LIN {X 0,Y 280.573,Z 825.158,A -85,B 0,C 180,E1 -18219.062,E2 -18219.062} C_VEL
LIN {X 0,Y 279.495,Z 836.896,A -85,B 0,C 180,E1 -18220.065,E2 -18220.065} C_VEL
LIN {X 0,Y 278.097,Z 847.663,A -85,B 0,C 180,E1 -18221.254,E2 -18221.254} C_VEL
LIN {X 0,Y 276.309,Z 858.858,A -85,B 0,C 180,E1 -18222.844,E2 -18222.844} C_VEL
LIN {X 0,Y 274.292,Z 869.192,A -85,B 0,C 180,E1 -18224.686,E2 -18224.686} C_VEL
LIN {X 0,Y 272.634,Z 876.745,A -85,B 0,C 180,E1 -18226.359,E2 -18226.359} C_VEL
LIN {X 0,Y 270.784,Z 884.275,A -85,B 0,C 180,E1 -18228.399,E2 -18228.399} C_VEL
LIN {X 0,Y 269.028,Z 890.984,A -85,B 0,C 180,E1 -18230.695,E2 -18230.695} C_VEL
LIN {X 0,Y 267.576,Z 895.963,A -85,B 0,C 180,E1 -18232.839,E2 -18232.839} C_VEL
LIN {X 0,Y 266.081,Z 900.757,A -85,B 0,C 180,E1 -18235.569,E2 -18235.569} C_VEL
LIN {X 0,Y 265.124,Z 903.749,A -85,B 0,C 180,E1 -18238.025,E2 -18238.025} C_VEL
LIN {X 0,Y 264.627,Z 905.127,A -85,B 0,C 180,E1 -18239.698,E2 -18239.698} C_VEL
LIN {X 0,Y 264.256,Z 906.046,A -85,B 0,C 180,E1 -18241.401,E2 -18241.401} C_VEL
LIN {X 0,Y 263.97,Z 906.49,A -85,B 0,C 180,E1 -18243.091,E2 -18243.091} C_VEL
LIN {X 0,Y 263.816,Z 906.395,A -85,B 0,C 180,E1 -18244.926,E2 -18244.926} C_VEL
LIN {X 0,Y 263.785,Z 905.92,A -85,B 0,C 180,E1 -18246.447,E2 -18246.447} C_VEL
LIN {X 0,Y 263.951,Z 904.438,A -85,B 0,C 180,E1 -18248.737,E2 -18248.737} C_VEL
LIN {X 0,Y 264.462,Z 901.575,A -85,B 0,C 180,E1 -18251.406,E2 -18251.406} C_VEL
LIN {X 0,Y 265.271,Z 897.734,A -85,B 0,C 180,E1 -18253.851,E2 -18253.851} C_VEL
LIN {X 0,Y 266.194,Z 892.722,A -85,B 0,C 180,E1 -18256.257,E2 -18256.257} C_VEL
LIN {X 0,Y 267.446,Z 886.349,A -85,B 0,C 180,E1 -18258.636,E2 -18258.636} C_VEL
LIN {X 0,Y 268.929,Z 878.429,A -85,B 0,C 180,E1 -18260.981,E2 -18260.981} C_VEL
LIN {X 0,Y 270.327,Z 870.307,A -85,B 0,C 180,E1 -18262.909,E2 -18262.909} C_VEL
LIN {X 0,Y 271.929,Z 860.358,A -85,B 0,C 180,E1 -18264.812,E2 -18264.812} C_VEL
LIN {X 0,Y 273.479,Z 849.327,A -85,B 0,C 180,E1 -18266.503,E2 -18266.503} C_VEL
LIN {X 0,Y 274.856,Z 837.273,A -85,B 0,C 180,E1 -18267.939,E2 -18267.939} C_VEL
LIN {X 0,Y 275.911,Z 824.671,A -85,B 0,C 180,E1 -18269.09,E2 -18269.09} C_VEL
LIN {X 0,Y 276.523,Z 812.385,A -85,B 0,C 180,E1 -18269.911,E2 -18269.911} C_VEL
LIN {X 0,Y 276.817,Z 798.91,A -85,B 0,C 180,E1 -18270.5,E2 -18270.5} C_VEL
LIN {X 0,Y 277.725,Z 751.411,A -85,B 0,C 180,E1 -18271.806,E2 -18271.806} C_VEL
LIN {X 0,Y 271.657,Z 736.963,A -85,B 0,C 180,E1 -18272.837,E2 -18272.837} C_VEL
LIN {X 0,Y 264.688,Z 722.978,A -85,B 0,C 180,E1 -18273.994,E2 -18273.994} C_VEL
LIN {X 0,Y 263.476,Z 720.392,A -85,B 0,C 180,E1 -18274.273,E2 -18274.273} C_VEL
LIN {X 0,Y 263.344,Z 719.73,A -85,B 0,C 180,E1 -18274.594,E2 -18274.594} C_VEL
LIN {X 0,Y 263.53,Z 719.652,A -85,B 0,C 180,E1 -18277.665,E2 -18277.665} C_VEL
LIN {X 0,Y 263.339,Z 719.672,A -85,B 0,C 180,E1 -18280.769,E2 -18280.769} C_VEL
LIN {X 0,Y 263.315,Z 719.673,A -85,B 0,C 180,E1 -18285.482,E2 -18285.482} C_VEL
LIN {X 0,Y 263.214,Z 719.678,A -85,B 0,C 180,E1 -18290.313,E2 -18290.313} C_VEL
LIN {X 0,Y 263.127,Z 719.691,A -85,B 0,C 180,E1 -18295.302,E2 -18295.302} C_VEL
LIN {X 0,Y 263.124,Z 719.7,A -85,B 0,C 180,E1 -18298.739,E2 -18298.739} C_VEL
LIN {X 0,Y 263.133,Z 719.698,A -85,B 0,C 180,E1 -18302.291,E2 -18302.291} C_VEL
LIN {X 0,Y 263.163,Z 719.673,A -85,B 0,C 180,E1 -18305.984,E2 -18305.984} C_VEL
LIN {X 0,Y 263.097,Z 719.713,A -85,B 0,C 180,E1 -18309.877,E2 -18309.877} C_VEL
LIN {X 0,Y 263.083,Z 719.716,A -85,B 0,C 180,E1 -18313.995,E2 -18313.995} C_VEL
LIN {X 0,Y 263.087,Z 719.713,A -85,B 0,C 180,E1 -18318.419,E2 -18318.419} C_VEL
LIN {X 0,Y 263.211,Z 719.896,A -85,B 0,C 180,E1 -18321.285,E2 -18321.285} C_VEL
LIN {X 0,Y 263.406,Z 720.866,A -85,B 0,C 180,E1 -18321.514,E2 -18321.514} C_VEL
LIN {X 0,Y 272.271,Z 746.098,A -85,B 0,C 180,E1 -18323.036,E2 -18323.036} C_VEL
LIN {X 0,Y 270.678,Z 798.339,A -85,B 0,C 180,E1 -18324.909,E2 -18324.909} C_VEL
LIN {X 0,Y 270.307,Z 809.826,A -85,B 0,C 180,E1 -18325.528,E2 -18325.528} C_VEL
LIN {X 0,Y 269.831,Z 820.372,A -85,B 0,C 180,E1 -18326.292,E2 -18326.292} C_VEL
LIN {X 0,Y 269.164,Z 830.302,A -85,B 0,C 180,E1 -18327.194,E2 -18327.194} C_VEL
LIN {X 0,Y 268.375,Z 841.093,A -85,B 0,C 180,E1 -18328.416,E2 -18328.416} C_VEL
LIN {X 0,Y 267.591,Z 849.983,A -85,B 0,C 180,E1 -18329.63,E2 -18329.63} C_VEL
LIN {X 0,Y 266.8,Z 858.729,A -85,B 0,C 180,E1 -18331.051,E2 -18331.051} C_VEL
LIN {X 0,Y 266.128,Z 866.2,A -85,B 0,C 180,E1 -18332.474,E2 -18332.474} C_VEL
LIN {X 0,Y 265.279,Z 874.154,A -85,B 0,C 180,E1 -18334.262,E2 -18334.262} C_VEL
LIN {X 0,Y 264.643,Z 881.015,A -85,B 0,C 180,E1 -18336.109,E2 -18336.109} C_VEL
LIN {X 0,Y 264.127,Z 887.251,A -85,B 0,C 180,E1 -18338.129,E2 -18338.129} C_VEL
LIN {X 0,Y 263.808,Z 891.489,A -85,B 0,C 180,E1 -18339.737,E2 -18339.737} C_VEL
LIN {X 0,Y 263.602,Z 894.43,A -85,B 0,C 180,E1 -18341.058,E2 -18341.058} C_VEL
LIN {X 0,Y 262.845,Z 896.919,A -85,B 0,C 180,E1 -18342.214,E2 -18342.214} C_VEL
LIN {X 0,Y 259.935,Z 900.48,A -85,B 0,C 180,E1 -18344.142,E2 -18344.142} C_VEL
LIN {X 0,Y 257.584,Z 902.751,A -85,B 0,C 180,E1 -18345.754,E2 -18345.754} C_VEL
LIN {X 0,Y 256.67,Z 904.09,A -85,B 0,C 180,E1 -18347.027,E2 -18347.027} C_VEL
LIN {X 0,Y 256.645,Z 904.457,A -85,B 0,C 180,E1 -18347.461,E2 -18347.461} C_VEL
LIN {X 0,Y 257.147,Z 906.07,A -85,B 0,C 180,E1 -18349.717,E2 -18349.717} C_VEL
LIN {X 0,Y 257.916,Z 906.726,A -85,B 0,C 180,E1 -18352.169,E2 -18352.169} C_VEL
LIN {X 0,Y 258.537,Z 906.558,A -85,B 0,C 180,E1 -18353.757,E2 -18353.757} C_VEL
LIN {X 0,Y 259.369,Z 905.964,A -85,B 0,C 180,E1 -18355.337,E2 -18355.337} C_VEL
LIN {X 0,Y 261.321,Z 903.482,A -85,B 0,C 180,E1 -18358.459,E2 -18358.459} C_VEL
LIN {X 0,Y 263.036,Z 900.45,A -85,B 0,C 180,E1 -18360.765,E2 -18360.765} C_VEL
LIN {X 0,Y 265.108,Z 896.26,A -85,B 0,C 180,E1 -18363.039,E2 -18363.039} C_VEL
LIN {X 0,Y 267.118,Z 891.825,A -85,B 0,C 180,E1 -18364.905,E2 -18364.905} C_VEL
LIN {X 0,Y 269.683,Z 885.252,A -85,B 0,C 180,E1 -18367.111,E2 -18367.111} C_VEL
LIN {X 0,Y 271.595,Z 880.039,A -85,B 0,C 180,E1 -18368.557,E2 -18368.557} C_VEL
LIN {X 0,Y 274.067,Z 872.242,A -85,B 0,C 180,E1 -18370.341,E2 -18370.341} C_VEL
LIN {X 0,Y 276.149,Z 864.832,A -85,B 0,C 180,E1 -18371.747,E2 -18371.747} C_VEL
LIN {X 0,Y 278.356,Z 856.069,A -85,B 0,C 180,E1 -18373.134,E2 -18373.134} C_VEL
LIN {X 0,Y 280.318,Z 846.92,A -85,B 0,C 180,E1 -18374.334,E2 -18374.334} C_VEL
LIN {X 0,Y 281.972,Z 837.469,A -85,B 0,C 180,E1 -18375.356,E2 -18375.356} C_VEL
LIN {X 0,Y 283.26,Z 827.918,A -85,B 0,C 180,E1 -18376.208,E2 -18376.208} C_VEL
LIN {X 0,Y 284.446,Z 816.78,A -85,B 0,C 180,E1 -18376.969,E2 -18376.969} C_VEL
LIN {X 0,Y 285.631,Z 800.883,A -85,B 0,C 180,E1 -18377.784,E2 -18377.784} C_VEL
LIN {X 0,Y 288.129,Z 773.827,A -85,B 0,C 180,E1 -18378.908,E2 -18378.908} C_VEL
LIN {X 0,Y 288.719,Z 767.247,A -85,B 0,C 180,E1 -18379.186,E2 -18379.186} C_VEL
LIN {X 0,Y 284.14,Z 758.529,A -85,B 0,C 180,E1 -18381.12,E2 -18381.12} C_VEL
LIN {X 0,Y 279.969,Z 751.63,A -85,B 0,C 180,E1 -18383.109,E2 -18383.109} C_VEL
LIN {X 0,Y 276.835,Z 747.044,A -85,B 0,C 180,E1 -18384.822,E2 -18384.822} C_VEL
LIN {X 0,Y 274.47,Z 743.25,A -85,B 0,C 180,E1 -18386.379,E2 -18386.379} C_VEL
LIN {X 0,Y 271.752,Z 740.074,A -85,B 0,C 180,E1 -18388.36,E2 -18388.36} C_VEL
LIN {X 0,Y 270.817,Z 738.098,A -85,B 0,C 180,E1 -18389.329,E2 -18389.329} C_VEL
LIN {X 0,Y 268.084,Z 735.681,A -85,B 0,C 180,E1 -18392.341,E2 -18392.341} C_VEL
LIN {X 0,Y 267.252,Z 733.95,A -85,B 0,C 180,E1 -18394.207,E2 -18394.207} C_VEL
LIN {X 0,Y 266.552,Z 733.96,A -85,B 0,C 180,E1 -18396.794,E2 -18396.794} C_VEL
LIN {X 0,Y 266.864,Z 735.363,A -85,B 0,C 180,E1 -18399.936,E2 -18399.936} C_VEL
LIN {X 0,Y 268.128,Z 737.207,A -85,B 0,C 180,E1 -18402.44,E2 -18402.44} C_VEL
LIN {X 0,Y 269.32,Z 739.283,A -85,B 0,C 180,E1 -18404.053,E2 -18404.053} C_VEL
LIN {X 0,Y 271.804,Z 742.654,A -85,B 0,C 180,E1 -18406.385,E2 -18406.385} C_VEL
LIN {X 0,Y 273.944,Z 746.353,A -85,B 0,C 180,E1 -18408.073,E2 -18408.073} C_VEL
LIN {X 0,Y 276.75,Z 755.997,A -85,B 0,C 180,E1 -18410.376,E2 -18410.376} C_VEL
LIN {X 0,Y 280.751,Z 769.642,A -85,B 0,C 180,E1 -18413.044,E2 -18413.044} C_VEL
LIN {X 0,Y 281.302,Z 772.583,A -85,B 0,C 180,E1 -18413.455,E2 -18413.455} C_VEL
LIN {X 0,Y 282.401,Z 792.767,A -85,B 0,C 180,E1 -18415.273,E2 -18415.273} C_VEL
LIN {X 0,Y 283.037,Z 812.394,A -85,B 0,C 180,E1 -18416.751,E2 -18416.751} C_VEL
LIN {X 0,Y 283.094,Z 822.192,A -85,B 0,C 180,E1 -18417.396,E2 -18417.396} C_VEL
LIN {X 0,Y 282.769,Z 841.316,A -85,B 0,C 180,E1 -18418.475,E2 -18418.475} C_VEL
LIN {X 0,Y 280.175,Z 867.058,A -85,B 0,C 180,E1 -18419.519,E2 -18419.519} C_VEL
LIN {X 0,Y 277.909,Z 882.038,A -85,B 0,C 180,E1 -18420.347,E2 -18420.347} C_VEL
LIN {X 0,Y 275.081,Z 895.368,A -85,B 0,C 180,E1 -18421.375,E2 -18421.375} C_VEL
LIN {X 0,Y 272.757,Z 905.306,A -85,B 0,C 180,E1 -18422.365,E2 -18422.365} C_VEL
LIN {X 0,Y 270.139,Z 915.057,A -85,B 0,C 180,E1 -18423.541,E2 -18423.541} C_VEL
LIN {X 0,Y 267.355,Z 924.567,A -85,B 0,C 180,E1 -18424.918,E2 -18424.918} C_VEL
LIN {X 0,Y 264.709,Z 933.598,A -85,B 0,C 180,E1 -18426.529,E2 -18426.529} C_VEL
LIN {X 0,Y 262.562,Z 940.532,A -85,B 0,C 180,E1 -18427.99,E2 -18427.99} C_VEL
LIN {X 0,Y 260.312,Z 948.007,A -85,B 0,C 180,E1 -18429.863,E2 -18429.863} C_VEL
LIN {X 0,Y 258.187,Z 955.518,A -85,B 0,C 180,E1 -18432.165,E2 -18432.165} C_VEL
LIN {X 0,Y 256.893,Z 960.781,A -85,B 0,C 180,E1 -18434.12,E2 -18434.12} C_VEL
LIN {X 0,Y 255.742,Z 965.991,A -85,B 0,C 180,E1 -18436.489,E2 -18436.489} C_VEL
LIN {X 0,Y 255.099,Z 970.126,A -85,B 0,C 180,E1 -18438.878,E2 -18438.878} C_VEL
LIN {X 0,Y 255.175,Z 976.468,A -85,B 0,C 180,E1 -18443.673,E2 -18443.673} C_VEL
LIN {X 0,Y 255.414,Z 978.203,A -85,B 0,C 180,E1 -18445.263,E2 -18445.263} C_VEL
LIN {X 0,Y 255.612,Z 979.494,A -85,B 0,C 180,E1 -18446.845,E2 -18446.845} C_VEL
LIN {X 0,Y 255.788,Z 980.353,A -85,B 0,C 180,E1 -18448.423,E2 -18448.423} C_VEL
LIN {X 0,Y 255.954,Z 980.742,A -85,B 0,C 180,E1 -18449.998,E2 -18449.998} C_VEL
LIN {X 0,Y 255.751,Z 980.652,A -85,B 0,C 180,E1 -18451.572,E2 -18451.572} C_VEL
LIN {X 0,Y 255.548,Z 980.148,A -85,B 0,C 180,E1 -18453.151,E2 -18453.151} C_VEL
LIN {X 0,Y 255.341,Z 979.232,A -85,B 0,C 180,E1 -18454.734,E2 -18454.734} C_VEL
LIN {X 0,Y 255.02,Z 976.923,A -85,B 0,C 180,E1 -18457.202,E2 -18457.202} C_VEL
LIN {X 0,Y 254.928,Z 973.806,A -85,B 0,C 180,E1 -18459.519,E2 -18459.519} C_VEL
LIN {X 0,Y 255.223,Z 969.585,A -85,B 0,C 180,E1 -18461.916,E2 -18461.916} C_VEL
LIN {X 0,Y 256.135,Z 963.256,A -85,B 0,C 180,E1 -18464.7,E2 -18464.7} C_VEL
LIN {X 0,Y 257.137,Z 957.383,A -85,B 0,C 180,E1 -18466.764,E2 -18466.764} C_VEL
LIN {X 0,Y 258.744,Z 951.013,A -85,B 0,C 180,E1 -18468.609,E2 -18468.609} C_VEL
LIN {X 0,Y 260.526,Z 943.101,A -85,B 0,C 180,E1 -18470.527,E2 -18470.527} C_VEL
LIN {X 0,Y 262.82,Z 933.587,A -85,B 0,C 180,E1 -18472.396,E2 -18472.396} C_VEL
LIN {X 0,Y 265.164,Z 923.078,A -85,B 0,C 180,E1 -18474.045,E2 -18474.045} C_VEL
LIN {X 0,Y 267.563,Z 911.507,A -85,B 0,C 180,E1 -18475.472,E2 -18475.472} C_VEL
LIN {X 0,Y 269.7,Z 899.511,A -85,B 0,C 180,E1 -18476.605,E2 -18476.605} C_VEL
LIN {X 0,Y 271.461,Z 886.354,A -85,B 0,C 180,E1 -18477.511,E2 -18477.511} C_VEL
LIN {X 0,Y 272.7,Z 872.76,A -85,B 0,C 180,E1 -18478.143,E2 -18478.143} C_VEL
LIN {X 0,Y 274.01,Z 835.757,A -85,B 0,C 180,E1 -18479.186,E2 -18479.186} C_VEL
LIN {X 0,Y 271.916,Z 808.359,A -85,B 0,C 180,E1 -18480.344,E2 -18480.344} C_VEL
LIN {X 0,Y 269.303,Z 784.538,A -85,B 0,C 180,E1 -18481.495,E2 -18481.495} C_VEL
LIN {X 0,Y 265.649,Z 760.465,A -85,B 0,C 180,E1 -18482.919,E2 -18482.919} C_VEL
LIN {X 0,Y 265.303,Z 757.226,A -85,B 0,C 180,E1 -18483.797,E2 -18483.797} C_VEL
LIN {X 0,Y 263.15,Z 746.364,A -85,B 0,C 180,E1 -18487.225,E2 -18487.225} C_VEL
LIN {X 0,Y 261.041,Z 737.55,A -85,B 0,C 180,E1 -18490.249,E2 -18490.249} C_VEL
LIN {X 0,Y 258.307,Z 728.035,A -85,B 0,C 180,E1 -18493.862,E2 -18493.862} C_VEL
LIN {X 0,Y 256.06,Z 720.679,A -85,B 0,C 180,E1 -18496.992,E2 -18496.992} C_VEL
LIN {X 0,Y 256.082,Z 720.572,A -85,B 0,C 180,E1 -18500.86,E2 -18500.86} C_VEL
LIN {X 0,Y 256.111,Z 720.561,A -85,B 0,C 180,E1 -18504.812,E2 -18504.812} C_VEL
LIN {X 0,Y 256.083,Z 720.582,A -85,B 0,C 180,E1 -18508.571,E2 -18508.571} C_VEL
LIN {X 0,Y 256.132,Z 720.575,A -85,B 0,C 180,E1 -18512.195,E2 -18512.195} C_VEL
LIN {X 0,Y 256.157,Z 720.571,A -85,B 0,C 180,E1 -18515.698,E2 -18515.698} C_VEL
LIN {X 0,Y 256.156,Z 720.568,A -85,B 0,C 180,E1 -18519.104,E2 -18519.104} C_VEL
LIN {X 0,Y 256.289,Z 720.559,A -85,B 0,C 180,E1 -18524.085,E2 -18524.085} C_VEL
LIN {X 0,Y 256.286,Z 720.561,A -85,B 0,C 180,E1 -18528.933,E2 -18528.933} C_VEL
LIN {X 0,Y 256.504,Z 720.524,A -85,B 0,C 180,E1 -18532.126,E2 -18532.126} C_VEL
LIN {X 0,Y 256.488,Z 720.528,A -85,B 0,C 180,E1 -18536.859,E2 -18536.859} C_VEL
LIN {X 0,Y 256.754,Z 720.491,A -85,B 0,C 180,E1 -18540,E2 -18540} C_VEL
LIN {X 0,Y 256.488,Z 720.533,A -85,B 0,C 180,E1 -18543.142,E2 -18543.142} C_VEL
LIN {X 0,Y 256.529,Z 720.524,A -85,B 0,C 180,E1 -18547.874,E2 -18547.874} C_VEL
LIN {X 0,Y 256.299,Z 720.558,A -85,B 0,C 180,E1 -18551.067,E2 -18551.067} C_VEL
LIN {X 0,Y 256.289,Z 720.552,A -85,B 0,C 180,E1 -18555.916,E2 -18555.916} C_VEL
LIN {X 0,Y 256.152,Z 720.58,A -85,B 0,C 180,E1 -18560.897,E2 -18560.897} C_VEL
LIN {X 0,Y 256.161,Z 720.563,A -85,B 0,C 180,E1 -18565.132,E2 -18565.132} C_VEL
LIN {X 0,Y 256.095,Z 720.573,A -85,B 0,C 180,E1 -18569.603,E2 -18569.603} C_VEL
LIN {X 0,Y 256.142,Z 720.825,A -85,B 0,C 180,E1 -18570.962,E2 -18570.962} C_VEL
LIN {X 0,Y 256.421,Z 721.972,A -85,B 0,C 180,E1 -18571.268,E2 -18571.268} C_VEL
LIN {X 0,Y 257.969,Z 724.576,A -85,B 0,C 180,E1 -18571.666,E2 -18571.666} C_VEL
LIN {X 0,Y 265.613,Z 736.935,A -85,B 0,C 180,E1 -18573.415,E2 -18573.415} C_VEL
LIN {X 0,Y 272.167,Z 749.03,A -85,B 0,C 180,E1 -18574.843,E2 -18574.843} C_VEL
LIN {X 0,Y 276.682,Z 758.44,A -85,B 0,C 180,E1 -18575.8,E2 -18575.8} C_VEL
LIN {X 0,Y 275.524,Z 798.704,A -85,B 0,C 180,E1 -18576.943,E2 -18576.943} C_VEL
LIN {X 0,Y 275.228,Z 812.621,A -85,B 0,C 180,E1 -18577.483,E2 -18577.483} C_VEL
LIN {X 0,Y 274.562,Z 825.156,A -85,B 0,C 180,E1 -18578.271,E2 -18578.271} C_VEL
LIN {X 0,Y 273.46,Z 836.856,A -85,B 0,C 180,E1 -18579.27,E2 -18579.27} C_VEL
LIN {X 0,Y 271.85,Z 848.731,A -85,B 0,C 180,E1 -18580.588,E2 -18580.588} C_VEL
LIN {X 0,Y 270.13,Z 859.173,A -85,B 0,C 180,E1 -18582.09,E2 -18582.09} C_VEL
LIN {X 0,Y 268.111,Z 869.167,A -85,B 0,C 180,E1 -18583.878,E2 -18583.878} C_VEL
LIN {X 0,Y 266.114,Z 877.902,A -85,B 0,C 180,E1 -18585.827,E2 -18585.827} C_VEL
LIN {X 0,Y 264.255,Z 885.108,A -85,B 0,C 180,E1 -18587.819,E2 -18587.819} C_VEL
LIN {X 0,Y 262.498,Z 891.489,A -85,B 0,C 180,E1 -18590.02,E2 -18590.02} C_VEL
LIN {X 0,Y 260.663,Z 897.444,A -85,B 0,C 180,E1 -18592.656,E2 -18592.656} C_VEL
LIN {X 0,Y 259.185,Z 901.88,A -85,B 0,C 180,E1 -18595.293,E2 -18595.293} C_VEL
LIN {X 0,Y 258.287,Z 904.526,A -85,B 0,C 180,E1 -18597.514,E2 -18597.514} C_VEL
LIN {X 0,Y 257.398,Z 906.79,A -85,B 0,C 180,E1 -18600.566,E2 -18600.566} C_VEL
LIN {X 0,Y 257.059,Z 907.387,A -85,B 0,C 180,E1 -18602.307,E2 -18602.307} C_VEL
LIN {X 0,Y 256.805,Z 907.46,A -85,B 0,C 180,E1 -18604.572,E2 -18604.572} C_VEL
LIN {X 0,Y 256.812,Z 906.365,A -85,B 0,C 180,E1 -18607.475,E2 -18607.475} C_VEL
LIN {X 0,Y 256.99,Z 905.107,A -85,B 0,C 180,E1 -18609.178,E2 -18609.178} C_VEL
LIN {X 0,Y 257.521,Z 902.294,A -85,B 0,C 180,E1 -18611.711,E2 -18611.711} C_VEL
LIN {X 0,Y 258.348,Z 898.358,A -85,B 0,C 180,E1 -18614.217,E2 -18614.217} C_VEL
LIN {X 0,Y 259.564,Z 892.259,A -85,B 0,C 180,E1 -18617.098,E2 -18617.098} C_VEL
LIN {X 0,Y 260.912,Z 885.535,A -85,B 0,C 180,E1 -18619.527,E2 -18619.527} C_VEL
LIN {X 0,Y 262.583,Z 876.743,A -85,B 0,C 180,E1 -18622.016,E2 -18622.016} C_VEL
LIN {X 0,Y 264.065,Z 868.503,A -85,B 0,C 180,E1 -18623.891,E2 -18623.891} C_VEL
LIN {X 0,Y 265.562,Z 859.122,A -85,B 0,C 180,E1 -18625.639,E2 -18625.639} C_VEL
LIN {X 0,Y 267.08,Z 848.303,A -85,B 0,C 180,E1 -18627.249,E2 -18627.249} C_VEL
LIN {X 0,Y 268.499,Z 835.993,A -85,B 0,C 180,E1 -18628.69,E2 -18628.69} C_VEL
LIN {X 0,Y 269.443,Z 824.479,A -85,B 0,C 180,E1 -18629.722,E2 -18629.722} C_VEL
LIN {X 0,Y 270.118,Z 811.171,A -85,B 0,C 180,E1 -18630.582,E2 -18630.582} C_VEL
LIN {X 0,Y 270.348,Z 798.125,A -85,B 0,C 180,E1 -18631.131,E2 -18631.131} C_VEL
LIN {X 0,Y 271.23,Z 753.034,A -85,B 0,C 180,E1 -18632.396,E2 -18632.396} C_VEL
LIN {X 0,Y 263.923,Z 736.114,A -85,B 0,C 180,E1 -18633.67,E2 -18633.67} C_VEL
LIN {X 0,Y 256.588,Z 721.779,A -85,B 0,C 180,E1 -18634.962,E2 -18634.962} C_VEL
LIN {X 0,Y 256.367,Z 720.699,A -85,B 0,C 180,E1 -18635.262,E2 -18635.262} C_VEL
LIN {X 0,Y 256.472,Z 720.532,A -85,B 0,C 180,E1 -18637.877,E2 -18637.877} C_VEL
LIN {X 0,Y 256.284,Z 720.551,A -85,B 0,C 180,E1 -18641.069,E2 -18641.069} C_VEL
LIN {X 0,Y 256.236,Z 720.558,A -85,B 0,C 180,E1 -18645.921,E2 -18645.921} C_VEL
LIN {X 0,Y 256.125,Z 720.566,A -85,B 0,C 180,E1 -18651.099,E2 -18651.099} C_VEL
LIN {X 0,Y 256.09,Z 720.569,A -85,B 0,C 180,E1 -18655.09,E2 -18655.09} C_VEL
LIN {X 0,Y 256.082,Z 720.576,A -85,B 0,C 180,E1 -18658.571,E2 -18658.571} C_VEL
LIN {X 0,Y 256.076,Z 720.581,A -85,B 0,C 180,E1 -18661.701,E2 -18661.701} C_VEL
LIN {X 0,Y 256.086,Z 720.548,A -85,B 0,C 180,E1 -18665.195,E2 -18665.195} C_VEL
LIN {X 0,Y 256.072,Z 720.586,A -85,B 0,C 180,E1 -18669.145,E2 -18669.145} C_VEL
LIN {X 0,Y 256.028,Z 720.594,A -85,B 0,C 180,E1 -18673.337,E2 -18673.337} C_VEL
LIN {X 0,Y 256.041,Z 720.593,A -85,B 0,C 180,E1 -18677.83,E2 -18677.83} C_VEL
LIN {X 0,Y 256.121,Z 720.79,A -85,B 0,C 180,E1 -18680.866,E2 -18680.866} C_VEL
LIN {X 0,Y 256.331,Z 721.653,A -85,B 0,C 180,E1 -18681.092,E2 -18681.092} C_VEL
LIN {X 0,Y 265.365,Z 747.332,A -85,B 0,C 180,E1 -18682.687,E2 -18682.687} C_VEL
LIN {X 0,Y 263.751,Z 799.297,A -85,B 0,C 180,E1 -18684.609,E2 -18684.609} C_VEL
LIN {X 0,Y 263.393,Z 810.483,A -85,B 0,C 180,E1 -18685.226,E2 -18685.226} C_VEL
LIN {X 0,Y 262.931,Z 820.543,A -85,B 0,C 180,E1 -18685.96,E2 -18685.96} C_VEL
LIN {X 0,Y 262.232,Z 830.761,A -85,B 0,C 180,E1 -18686.902,E2 -18686.902} C_VEL
LIN {X 0,Y 261.4,Z 841.61,A -85,B 0,C 180,E1 -18688.154,E2 -18688.154} C_VEL
LIN {X 0,Y 260.624,Z 850.368,A -85,B 0,C 180,E1 -18689.369,E2 -18689.369} C_VEL
LIN {X 0,Y 259.776,Z 859.362,A -85,B 0,C 180,E1 -18690.858,E2 -18690.858} C_VEL
LIN {X 0,Y 258.975,Z 867.829,A -85,B 0,C 180,E1 -18692.526,E2 -18692.526} C_VEL
LIN {X 0,Y 258.217,Z 874.992,A -85,B 0,C 180,E1 -18694.184,E2 -18694.184} C_VEL
LIN {X 0,Y 257.62,Z 881.147,A -85,B 0,C 180,E1 -18695.844,E2 -18695.844} C_VEL
LIN {X 0,Y 257.061,Z 887.939,A -85,B 0,C 180,E1 -18698.06,E2 -18698.06} C_VEL
LIN {X 0,Y 256.691,Z 892.865,A -85,B 0,C 180,E1 -18699.986,E2 -18699.986} C_VEL
LIN {X 0,Y 256.472,Z 896.444,A -85,B 0,C 180,E1 -18701.631,E2 -18701.631} C_VEL
LIN {X 0,Y 256.382,Z 900.642,A -85,B 0,C 180,E1 -18704.09,E2 -18704.09} C_VEL
LIN {X 0,Y 256.422,Z 902.739,A -85,B 0,C 180,E1 -18705.719,E2 -18705.719} C_VEL
LIN {X 0,Y 256.645,Z 904.457,A -85,B 0,C 180,E1 -18707.461,E2 -18707.461} C_VEL
LIN {X 0,Y 256.215,Z 905.627,A -85,B 0,C 180,E1 -18708.758,E2 -18708.758} C_VEL
LIN {X 0,Y 253.941,Z 907.038,A -85,B 0,C 180,E1 -18710.903,E2 -18710.903} C_VEL
LIN {X 0,Y 251.911,Z 907.826,A -85,B 0,C 180,E1 -18713.096,E2 -18713.096} C_VEL
LIN {X 0,Y 251.868,Z 907.665,A -85,B 0,C 180,E1 -18714.44,E2 -18714.44} C_VEL
LIN {X 0,Y 253.362,Z 906.546,A -85,B 0,C 180,E1 -18717.006,E2 -18717.006} C_VEL
LIN {X 0,Y 254.318,Z 905.473,A -85,B 0,C 180,E1 -18718.416,E2 -18718.416} C_VEL
LIN {X 0,Y 256.11,Z 902.774,A -85,B 0,C 180,E1 -18720.786,E2 -18720.786} C_VEL
LIN {X 0,Y 258.263,Z 898.978,A -85,B 0,C 180,E1 -18723.12,E2 -18723.12} C_VEL
LIN {X 0,Y 260.865,Z 893.783,A -85,B 0,C 180,E1 -18725.488,E2 -18725.488} C_VEL
LIN {X 0,Y 263.483,Z 887.618,A -85,B 0,C 180,E1 -18727.664,E2 -18727.664} C_VEL
LIN {X 0,Y 265.985,Z 881.112,A -85,B 0,C 180,E1 -18729.505,E2 -18729.505} C_VEL
LIN {X 0,Y 268.656,Z 873.339,A -85,B 0,C 180,E1 -18731.315,E2 -18731.315} C_VEL
LIN {X 0,Y 271.182,Z 864.946,A -85,B 0,C 180,E1 -18732.916,E2 -18732.916} C_VEL
LIN {X 0,Y 273.248,Z 857.186,A -85,B 0,C 180,E1 -18734.143,E2 -18734.143} C_VEL
LIN {X 0,Y 275.313,Z 847.977,A -85,B 0,C 180,E1 -18735.358,E2 -18735.358} C_VEL
LIN {X 0,Y 277.107,Z 838.593,A -85,B 0,C 180,E1 -18736.389,E2 -18736.389} C_VEL
LIN {X 0,Y 278.498,Z 829.176,A -85,B 0,C 180,E1 -18737.248,E2 -18737.248} C_VEL
LIN {X 0,Y 279.725,Z 818.882,A -85,B 0,C 180,E1 -18737.972,E2 -18737.972} C_VEL
LIN {X 0,Y 280.834,Z 805.286,A -85,B 0,C 180,E1 -18738.701,E2 -18738.701} C_VEL
LIN {X 0,Y 283.663,Z 775.908,A -85,B 0,C 180,E1 -18739.978,E2 -18739.978} C_VEL
LIN {X 0,Y 284.261,Z 770.773,A -85,B 0,C 180,E1 -18740.178,E2 -18740.178} C_VEL
LIN {X 0,Y 280.643,Z 763.677,A -85,B 0,C 180,E1 -18741.85,E2 -18741.85} C_VEL
LIN {X 0,Y 277.078,Z 757.516,A -85,B 0,C 180,E1 -18743.69,E2 -18743.69} C_VEL
LIN {X 0,Y 274.185,Z 753.127,A -85,B 0,C 180,E1 -18745.385,E2 -18745.385} C_VEL
LIN {X 0,Y 271.891,Z 749.383,A -85,B 0,C 180,E1 -18747.001,E2 -18747.001} C_VEL
LIN {X 0,Y 269.645,Z 746.491,A -85,B 0,C 180,E1 -18748.809,E2 -18748.809} C_VEL
LIN {X 0,Y 269.001,Z 744.934,A -85,B 0,C 180,E1 -18749.547,E2 -18749.547} C_VEL
LIN {X 0,Y 266.327,Z 742.326,A -85,B 0,C 180,E1 -18752.749,E2 -18752.749} C_VEL
LIN {X 0,Y 265.649,Z 740.82,A -85,B 0,C 180,E1 -18754.442,E2 -18754.442} C_VEL
LIN {X 0,Y 265.022,Z 741.066,A -85,B 0,C 180,E1 -18757.289,E2 -18757.289} C_VEL
LIN {X 0,Y 265.658,Z 742.812,A -85,B 0,C 180,E1 -18760.691,E2 -18760.691} C_VEL
LIN {X 0,Y 266.791,Z 744.529,A -85,B 0,C 180,E1 -18762.703,E2 -18762.703} C_VEL
LIN {X 0,Y 269.755,Z 749.236,A -85,B 0,C 180,E1 -18766.02,E2 -18766.02} C_VEL
LIN {X 0,Y 271.418,Z 752.365,A -85,B 0,C 180,E1 -18767.446,E2 -18767.446} C_VEL
LIN {X 0,Y 273.757,Z 761.549,A -85,B 0,C 180,E1 -18769.668,E2 -18769.668} C_VEL
LIN {X 0,Y 277.291,Z 774.611,A -85,B 0,C 180,E1 -18772.269,E2 -18772.269} C_VEL
LIN {X 0,Y 277.724,Z 783.67,A -85,B 0,C 180,E1 -18773.177,E2 -18773.177} C_VEL
LIN {X 0,Y 278.338,Z 800.839,A -85,B 0,C 180,E1 -18774.683,E2 -18774.683} C_VEL
LIN {X 0,Y 278.608,Z 820.03,A -85,B 0,C 180,E1 -18776.124,E2 -18776.124} C_VEL
LIN {X 0,Y 277.967,Z 842.031,A -85,B 0,C 180,E1 -18777.421,E2 -18777.421} C_VEL
LIN {X 0,Y 275.276,Z 866.945,A -85,B 0,C 180,E1 -18778.455,E2 -18778.455} C_VEL
LIN {X 0,Y 272.827,Z 881.537,A -85,B 0,C 180,E1 -18779.309,E2 -18779.309} C_VEL
LIN {X 0,Y 270.31,Z 892.792,A -85,B 0,C 180,E1 -18780.18,E2 -18780.18} C_VEL
LIN {X 0,Y 267.354,Z 904.35,A -85,B 0,C 180,E1 -18781.329,E2 -18781.329} C_VEL
LIN {X 0,Y 264.632,Z 914.026,A -85,B 0,C 180,E1 -18782.518,E2 -18782.518} C_VEL
LIN {X 0,Y 261.725,Z 923.396,A -85,B 0,C 180,E1 -18783.912,E2 -18783.912} C_VEL
LIN {X 0,Y 259.443,Z 930.525,A -85,B 0,C 180,E1 -18785.171,E2 -18785.171} C_VEL
LIN {X 0,Y 256.529,Z 939.269,A -85,B 0,C 180,E1 -18787.018,E2 -18787.018} C_VEL
LIN {X 0,Y 254.103,Z 946.708,A -85,B 0,C 180,E1 -18788.925,E2 -18788.925} C_VEL
LIN {X 0,Y 252.097,Z 953.057,A -85,B 0,C 180,E1 -18790.876,E2 -18790.876} C_VEL
LIN {X 0,Y 250.205,Z 959.359,A -85,B 0,C 180,E1 -18793.228,E2 -18793.228} C_VEL
LIN {X 0,Y 249.101,Z 963.911,A -85,B 0,C 180,E1 -18795.288,E2 -18795.288} C_VEL
LIN {X 0,Y 248.237,Z 968.217,A -85,B 0,C 180,E1 -18797.738,E2 -18797.738} C_VEL
LIN {X 0,Y 247.966,Z 971.544,A -85,B 0,C 180,E1 -18800.207,E2 -18800.207} C_VEL
LIN {X 0,Y 248.085,Z 974.096,A -85,B 0,C 180,E1 -18802.531,E2 -18802.531} C_VEL
LIN {X 0,Y 248.342,Z 977.114,A -85,B 0,C 180,E1 -18805.127,E2 -18805.127} C_VEL
LIN {X 0,Y 248.552,Z 978.423,A -85,B 0,C 180,E1 -18806.756,E2 -18806.756} C_VEL
LIN {X 0,Y 248.745,Z 979.303,A -85,B 0,C 180,E1 -18808.379,E2 -18808.379} C_VEL
LIN {X 0,Y 248.921,Z 979.722,A -85,B 0,C 180,E1 -18809.998,E2 -18809.998} C_VEL
LIN {X 0,Y 248.704,Z 979.642,A -85,B 0,C 180,E1 -18811.617,E2 -18811.617} C_VEL
LIN {X 0,Y 248.491,Z 979.15,A -85,B 0,C 180,E1 -18813.24,E2 -18813.24} C_VEL
LIN {X 0,Y 248.271,Z 978.247,A -85,B 0,C 180,E1 -18814.869,E2 -18814.869} C_VEL
LIN {X 0,Y 247.951,Z 976.151,A -85,B 0,C 180,E1 -18817.229,E2 -18817.229} C_VEL
LIN {X 0,Y 247.861,Z 972.884,A -85,B 0,C 180,E1 -18819.793,E2 -18819.793} C_VEL
LIN {X 0,Y 248.217,Z 968.702,A -85,B 0,C 180,E1 -18822.258,E2 -18822.258} C_VEL
LIN {X 0,Y 249.212,Z 962.431,A -85,B 0,C 180,E1 -18825.118,E2 -18825.118} C_VEL
LIN {X 0,Y 250.656,Z 955.515,A -85,B 0,C 180,E1 -18827.578,E2 -18827.578} C_VEL
LIN {X 0,Y 252.655,Z 947.278,A -85,B 0,C 180,E1 -18829.92,E2 -18829.92} C_VEL
LIN {X 0,Y 254.777,Z 938.851,A -85,B 0,C 180,E1 -18831.861,E2 -18831.861} C_VEL
LIN {X 0,Y 257.306,Z 928.674,A -85,B 0,C 180,E1 -18833.756,E2 -18833.756} C_VEL
LIN {X 0,Y 259.906,Z 917.264,A -85,B 0,C 180,E1 -18835.418,E2 -18835.418} C_VEL
LIN {X 0,Y 262.2,Z 906.175,A -85,B 0,C 180,E1 -18836.675,E2 -18836.675} C_VEL
LIN {X 0,Y 264.255,Z 893.986,A -85,B 0,C 180,E1 -18837.735,E2 -18837.735} C_VEL
LIN {X 0,Y 265.807,Z 881.438,A -85,B 0,C 180,E1 -18838.526,E2 -18838.526} C_VEL
LIN {X 0,Y 266.809,Z 868.435,A -85,B 0,C 180,E1 -18839.065,E2 -18839.065} C_VEL
LIN {X 0,Y 267.971,Z 836.435,A -85,B 0,C 180,E1 -18839.968,E2 -18839.968} C_VEL
LIN {X 0,Y 266.023,Z 809.893,A -85,B 0,C 180,E1 -18841.123,E2 -18841.123} C_VEL
LIN {X 0,Y 263.553,Z 786.25,A -85,B 0,C 180,E1 -18842.301,E2 -18842.301} C_VEL
LIN {X 0,Y 259.87,Z 762.613,A -85,B 0,C 180,E1 -18843.721,E2 -18843.721} C_VEL
LIN {X 0,Y 258.562,Z 759.035,A -85,B 0,C 180,E1 -18844.141,E2 -18844.141} C_VEL
LIN {X 0,Y 256.829,Z 749.961,A -85,B 0,C 180,E1 -18847.011,E2 -18847.011} C_VEL
LIN {X 0,Y 254.791,Z 741.269,A -85,B 0,C 180,E1 -18850.054,E2 -18850.054} C_VEL
LIN {X 0,Y 252.241,Z 732.147,A -85,B 0,C 180,E1 -18853.58,E2 -18853.58} C_VEL
LIN {X 0,Y 249.818,Z 724.085,A -85,B 0,C 180,E1 -18857.004,E2 -18857.004} C_VEL
LIN {X 0,Y 249.025,Z 721.503,A -85,B 0,C 180,E1 -18858.319,E2 -18858.319} C_VEL
LIN {X 0,Y 249.047,Z 721.464,A -85,B 0,C 180,E1 -18862.195,E2 -18862.195} C_VEL
LIN {X 0,Y 249.052,Z 721.444,A -85,B 0,C 180,E1 -18865.641,E2 -18865.641} C_VEL
LIN {X 0,Y 249.042,Z 721.461,A -85,B 0,C 180,E1 -18869.472,E2 -18869.472} C_VEL
LIN {X 0,Y 249.064,Z 721.461,A -85,B 0,C 180,E1 -18873.161,E2 -18873.161} C_VEL
LIN {X 0,Y 249.069,Z 721.46,A -85,B 0,C 180,E1 -18876.732,E2 -18876.732} C_VEL
LIN {X 0,Y 249.101,Z 721.456,A -85,B 0,C 180,E1 -18880.211,E2 -18880.211} C_VEL
LIN {X 0,Y 249.231,Z 721.433,A -85,B 0,C 180,E1 -18883.621,E2 -18883.621} C_VEL
LIN {X 0,Y 249.233,Z 721.44,A -85,B 0,C 180,E1 -18888.616,E2 -18888.616} C_VEL
LIN {X 0,Y 249.443,Z 721.402,A -85,B 0,C 180,E1 -18891.902,E2 -18891.902} C_VEL
LIN {X 0,Y 249.286,Z 721.422,A -85,B 0,C 180,E1 -18895.149,E2 -18895.149} C_VEL
LIN {X 0,Y 249.665,Z 721.385,A -85,B 0,C 180,E1 -18898.387,E2 -18898.387} C_VEL
LIN {X 0,Y 249.665,Z 721.382,A -85,B 0,C 180,E1 -18901.613,E2 -18901.613} C_VEL
LIN {X 0,Y 249.437,Z 721.41,A -85,B 0,C 180,E1 -18906.832,E2 -18906.832} C_VEL
LIN {X 0,Y 249.378,Z 721.417,A -85,B 0,C 180,E1 -18909.735,E2 -18909.735} C_VEL
LIN {X 0,Y 249.195,Z 721.443,A -85,B 0,C 180,E1 -18914.704,E2 -18914.704} C_VEL
LIN {X 0,Y 249.128,Z 721.453,A -85,B 0,C 180,E1 -18918.079,E2 -18918.079} C_VEL
LIN {X 0,Y 249.074,Z 721.453,A -85,B 0,C 180,E1 -18921.52,E2 -18921.52} C_VEL
LIN {X 0,Y 249.108,Z 721.446,A -85,B 0,C 180,E1 -18925.477,E2 -18925.477} C_VEL
LIN {X 0,Y 249.081,Z 721.653,A -85,B 0,C 180,E1 -18929.59,E2 -18929.59} C_VEL
LIN {X 0,Y 249.282,Z 722.562,A -85,B 0,C 180,E1 -18929.913,E2 -18929.913} C_VEL
LIN {X 0,Y 250.807,Z 725.315,A -85,B 0,C 180,E1 -18930.349,E2 -18930.349} C_VEL
LIN {X 0,Y 251.877,Z 726.635,A -85,B 0,C 180,E1 -18930.612,E2 -18930.612} C_VEL
LIN {X 0,Y 260.84,Z 741.279,A -85,B 0,C 180,E1 -18932.78,E2 -18932.78} C_VEL
LIN {X 0,Y 267.439,Z 753.655,A -85,B 0,C 180,E1 -18934.289,E2 -18934.289} C_VEL
LIN {X 0,Y 270.712,Z 760.629,A -85,B 0,C 180,E1 -18935.018,E2 -18935.018} C_VEL
LIN {X 0,Y 269.543,Z 800.865,A -85,B 0,C 180,E1 -18936.192,E2 -18936.192} C_VEL
LIN {X 0,Y 269.225,Z 814.153,A -85,B 0,C 180,E1 -18936.738,E2 -18936.738} C_VEL
LIN {X 0,Y 268.448,Z 827.058,A -85,B 0,C 180,E1 -18937.577,E2 -18937.577} C_VEL
LIN {X 0,Y 267.242,Z 838.918,A -85,B 0,C 180,E1 -18938.631,E2 -18938.631} C_VEL
LIN {X 0,Y 265.667,Z 849.949,A -85,B 0,C 180,E1 -18939.904,E2 -18939.904} C_VEL
LIN {X 0,Y 263.797,Z 860.58,A -85,B 0,C 180,E1 -18941.474,E2 -18941.474} C_VEL
LIN {X 0,Y 261.739,Z 870.271,A -85,B 0,C 180,E1 -18943.256,E2 -18943.256} C_VEL
LIN {X 0,Y 259.613,Z 879.06,A -85,B 0,C 180,E1 -18945.267,E2 -18945.267} C_VEL
LIN {X 0,Y 257.326,Z 887.337,A -85,B 0,C 180,E1 -18947.664,E2 -18947.664} C_VEL
LIN {X 0,Y 255.657,Z 893.088,A -85,B 0,C 180,E1 -18949.758,E2 -18949.758} C_VEL
LIN {X 0,Y 253.752,Z 898.928,A -85,B 0,C 180,E1 -18952.463,E2 -18952.463} C_VEL
LIN {X 0,Y 252.22,Z 903.233,A -85,B 0,C 180,E1 -18955.168,E2 -18955.168} C_VEL
LIN {X 0,Y 251.132,Z 906.17,A -85,B 0,C 180,E1 -18957.881,E2 -18957.881} C_VEL
LIN {X 0,Y 250.415,Z 907.861,A -85,B 0,C 180,E1 -18960.463,E2 -18960.463} C_VEL
LIN {X 0,Y 249.898,Z 908.546,A -85,B 0,C 180,E1 -18963.261,E2 -18963.261} C_VEL
LIN {X 0,Y 249.749,Z 908.386,A -85,B 0,C 180,E1 -18965.035,E2 -18965.035} C_VEL
LIN {X 0,Y 249.835,Z 906.916,A -85,B 0,C 180,E1 -18968.174,E2 -18968.174} C_VEL
LIN {X 0,Y 250.33,Z 904.092,A -85,B 0,C 180,E1 -18971.167,E2 -18971.167} C_VEL
LIN {X 0,Y 251.142,Z 900.443,A -85,B 0,C 180,E1 -18973.752,E2 -18973.752} C_VEL
LIN {X 0,Y 252.132,Z 895.645,A -85,B 0,C 180,E1 -18976.298,E2 -18976.298} C_VEL
LIN {X 0,Y 253.418,Z 889.506,A -85,B 0,C 180,E1 -18978.809,E2 -18978.809} C_VEL
LIN {X 0,Y 255.027,Z 881.534,A -85,B 0,C 180,E1 -18981.364,E2 -18981.364} C_VEL
LIN {X 0,Y 256.782,Z 872.255,A -85,B 0,C 180,E1 -18983.717,E2 -18983.717} C_VEL
LIN {X 0,Y 258.515,Z 862.29,A -85,B 0,C 180,E1 -18985.715,E2 -18985.715} C_VEL
LIN {X 0,Y 260.166,Z 851.439,A -85,B 0,C 180,E1 -18987.458,E2 -18987.458} C_VEL
LIN {X 0,Y 261.537,Z 840.484,A -85,B 0,C 180,E1 -18988.847,E2 -18988.847} C_VEL
LIN {X 0,Y 262.742,Z 827.673,A -85,B 0,C 180,E1 -18990.098,E2 -18990.098} C_VEL
LIN {X 0,Y 263.489,Z 815.066,A -85,B 0,C 180,E1 -18991.005,E2 -18991.005} C_VEL
LIN {X 0,Y 263.859,Z 801.921,A -85,B 0,C 180,E1 -18991.625,E2 -18991.625} C_VEL
LIN {X 0,Y 264.78,Z 754.831,A -85,B 0,C 180,E1 -18992.998,E2 -18992.998} C_VEL
LIN {X 0,Y 257.623,Z 738.43,A -85,B 0,C 180,E1 -18994.292,E2 -18994.292} C_VEL
LIN {X 0,Y 249.537,Z 722.367,A -85,B 0,C 180,E1 -18995.811,E2 -18995.811} C_VEL
LIN {X 0,Y 249.4,Z 721.487,A -85,B 0,C 180,E1 -18996.17,E2 -18996.17} C_VEL
LIN {X 0,Y 249.337,Z 721.42,A -85,B 0,C 180,E1 -18999.739,E2 -18999.739} C_VEL
LIN {X 0,Y 249.176,Z 721.432,A -85,B 0,C 180,E1 -19004.707,E2 -19004.707} C_VEL
LIN {X 0,Y 249.091,Z 721.454,A -85,B 0,C 180,E1 -19008.083,E2 -19008.083} C_VEL
LIN {X 0,Y 249.049,Z 721.452,A -85,B 0,C 180,E1 -19011.524,E2 -19011.524} C_VEL
LIN {X 0,Y 249.051,Z 721.441,A -85,B 0,C 180,E1 -19015.442,E2 -19015.442} C_VEL
LIN {X 0,Y 249.03,Z 721.457,A -85,B 0,C 180,E1 -19018.97,E2 -19018.97} C_VEL
LIN {X 0,Y 249.033,Z 721.45,A -85,B 0,C 180,E1 -19022.428,E2 -19022.428} C_VEL
LIN {X 0,Y 249.02,Z 721.437,A -85,B 0,C 180,E1 -19026.35,E2 -19026.35} C_VEL
LIN {X 0,Y 248.985,Z 721.469,A -85,B 0,C 180,E1 -19030.485,E2 -19030.485} C_VEL
LIN {X 0,Y 248.969,Z 721.472,A -85,B 0,C 180,E1 -19034.89,E2 -19034.89} C_VEL
LIN {X 0,Y 248.987,Z 721.47,A -85,B 0,C 180,E1 -19037.356,E2 -19037.356} C_VEL
LIN {X 0,Y 249.061,Z 721.673,A -85,B 0,C 180,E1 -19040.42,E2 -19040.42} C_VEL
LIN {X 0,Y 249.311,Z 722.677,A -85,B 0,C 180,E1 -19040.668,E2 -19040.668} C_VEL
LIN {X 0,Y 258.373,Z 748.6,A -85,B 0,C 180,E1 -19042.318,E2 -19042.318} C_VEL
LIN {X 0,Y 256.824,Z 800.262,A -85,B 0,C 180,E1 -19044.322,E2 -19044.322} C_VEL
LIN {X 0,Y 256.446,Z 811.52,A -85,B 0,C 180,E1 -19044.965,E2 -19044.965} C_VEL
LIN {X 0,Y 255.788,Z 823.152,A -85,B 0,C 180,E1 -19045.861,E2 -19045.861} C_VEL
LIN {X 0,Y 255.114,Z 832.814,A -85,B 0,C 180,E1 -19046.802,E2 -19046.802} C_VEL
LIN {X 0,Y 254.429,Z 841.918,A -85,B 0,C 180,E1 -19047.877,E2 -19047.877} C_VEL
LIN {X 0,Y 253.533,Z 851.554,A -85,B 0,C 180,E1 -19049.245,E2 -19049.245} C_VEL
LIN {X 0,Y 252.755,Z 859.908,A -85,B 0,C 180,E1 -19050.654,E2 -19050.654} C_VEL
LIN {X 0,Y 252.033,Z 867.524,A -85,B 0,C 180,E1 -19052.155,E2 -19052.155} C_VEL
LIN {X 0,Y 251.249,Z 874.922,A -85,B 0,C 180,E1 -19053.86,E2 -19053.86} C_VEL
LIN {X 0,Y 250.504,Z 882.618,A -85,B 0,C 180,E1 -19055.995,E2 -19055.995} C_VEL
LIN {X 0,Y 249.969,Z 888.93,A -85,B 0,C 180,E1 -19058.101,E2 -19058.101} C_VEL
LIN {X 0,Y 249.563,Z 894.243,A -85,B 0,C 180,E1 -19060.249,E2 -19060.249} C_VEL
LIN {X 0,Y 249.394,Z 897.792,A -85,B 0,C 180,E1 -19061.941,E2 -19061.941} C_VEL
LIN {X 0,Y 249.339,Z 901.924,A -85,B 0,C 180,E1 -19064.468,E2 -19064.468} C_VEL
LIN {X 0,Y 249.601,Z 905.345,A -85,B 0,C 180,E1 -19067.479,E2 -19067.479} C_VEL
LIN {X 0,Y 250.276,Z 907.334,A -85,B 0,C 180,E1 -19070.3,E2 -19070.3} C_VEL
LIN {X 0,Y 250.8,Z 907.827,A -85,B 0,C 180,E1 -19071.945,E2 -19071.945} C_VEL
LIN {X 0,Y 251.868,Z 907.665,A -85,B 0,C 180,E1 -19074.44,E2 -19074.44} C_VEL
LIN {X 0,Y 251.926,Z 907.428,A -85,B 0,C 180,E1 -19075.78,E2 -19075.78} C_VEL
LIN {X 0,Y 250.5,Z 906.669,A -85,B 0,C 180,E1 -19078.01,E2 -19078.01} C_VEL
LIN {X 0,Y 249.435,Z 905.731,A -85,B 0,C 180,E1 -19079.799,E2 -19079.799} C_VEL
LIN {X 0,Y 249.516,Z 904.526,A -85,B 0,C 180,E1 -19081.131,E2 -19081.131} C_VEL
LIN {X 0,Y 249.819,Z 904.044,A -85,B 0,C 180,E1 -19081.565,E2 -19081.565} C_VEL
LIN {X 0,Y 252.193,Z 900.202,A -85,B 0,C 180,E1 -19083.995,E2 -19083.995} C_VEL
LIN {X 0,Y 255.428,Z 894.005,A -85,B 0,C 180,E1 -19086.762,E2 -19086.762} C_VEL
LIN {X 0,Y 257.811,Z 888.809,A -85,B 0,C 180,E1 -19088.623,E2 -19088.623} C_VEL
LIN {X 0,Y 260.524,Z 882.35,A -85,B 0,C 180,E1 -19090.491,E2 -19090.491} C_VEL
LIN {X 0,Y 263.382,Z 874.548,A -85,B 0,C 180,E1 -19092.326,E2 -19092.326} C_VEL
LIN {X 0,Y 266.059,Z 866.148,A -85,B 0,C 180,E1 -19093.948,E2 -19093.948} C_VEL
LIN {X 0,Y 268.276,Z 858.466,A -85,B 0,C 180,E1 -19095.187,E2 -19095.187} C_VEL
LIN {X 0,Y 270.173,Z 850.835,A -85,B 0,C 180,E1 -19096.238,E2 -19096.238} C_VEL
LIN {X 0,Y 272.393,Z 839.993,A -85,B 0,C 180,E1 -19097.454,E2 -19097.454} C_VEL
LIN {X 0,Y 273.939,Z 830.122,A -85,B 0,C 180,E1 -19098.356,E2 -19098.356} C_VEL
LIN {X 0,Y 275.274,Z 819.778,A -85,B 0,C 180,E1 -19099.094,E2 -19099.094} C_VEL
LIN {X 0,Y 276.661,Z 804.387,A -85,B 0,C 180,E1 -19099.927,E2 -19099.927} C_VEL
LIN {X 0,Y 279.735,Z 775.429,A -85,B 0,C 180,E1 -19101.196,E2 -19101.196} C_VEL
LIN {X 0,Y 279.828,Z 774.049,A -85,B 0,C 180,E1 -19101.277,E2 -19101.277} C_VEL
LIN {X 0,Y 276.185,Z 766.767,A -85,B 0,C 180,E1 -19103.172,E2 -19103.172} C_VEL
LIN {X 0,Y 273.296,Z 762.013,A -85,B 0,C 180,E1 -19104.825,E2 -19104.825} C_VEL
LIN {X 0,Y 271.737,Z 759.397,A -85,B 0,C 180,E1 -19105.86,E2 -19105.86} C_VEL
LIN {X 0,Y 269.72,Z 755.934,A -85,B 0,C 180,E1 -19107.384,E2 -19107.384} C_VEL
LIN {X 0,Y 267.506,Z 752.826,A -85,B 0,C 180,E1 -19109.325,E2 -19109.325} C_VEL
LIN {X 0,Y 266.904,Z 751.55,A -85,B 0,C 180,E1 -19110.02,E2 -19110.02} C_VEL
LIN {X 0,Y 264.569,Z 748.927,A -85,B 0,C 180,E1 -19113.207,E2 -19113.207} C_VEL
LIN {X 0,Y 264.129,Z 747.782,A -85,B 0,C 180,E1 -19114.423,E2 -19114.423} C_VEL
LIN {X 0,Y 263.534,Z 747.864,A -85,B 0,C 180,E1 -19116.862,E2 -19116.862} C_VEL
LIN {X 0,Y 263.921,Z 749.435,A -85,B 0,C 180,E1 -19120.218,E2 -19120.218} C_VEL
LIN {X 0,Y 265.171,Z 751.486,A -85,B 0,C 180,E1 -19122.614,E2 -19122.614} C_VEL
LIN {X 0,Y 267.696,Z 755.781,A -85,B 0,C 180,E1 -19125.617,E2 -19125.617} C_VEL
LIN {X 0,Y 268.984,Z 758.448,A -85,B 0,C 180,E1 -19126.827,E2 -19126.827} C_VEL
LIN {X 0,Y 270.839,Z 766.697,A -85,B 0,C 180,E1 -19128.847,E2 -19128.847} C_VEL
LIN {X 0,Y 273.71,Z 778.773,A -85,B 0,C 180,E1 -19131.326,E2 -19131.326} C_VEL
LIN {X 0,Y 274.155,Z 798.605,A -85,B 0,C 180,E1 -19133.209,E2 -19133.209} C_VEL
LIN {X 0,Y 274.23,Z 820.221,A -85,B 0,C 180,E1 -19134.919,E2 -19134.919} C_VEL
LIN {X 0,Y 273.394,Z 842.789,A -85,B 0,C 180,E1 -19136.309,E2 -19136.309} C_VEL
LIN {X 0,Y 270.815,Z 864.97,A -85,B 0,C 180,E1 -19137.251,E2 -19137.251} C_VEL
LIN {X 0,Y 268.048,Z 880.248,A -85,B 0,C 180,E1 -19138.15,E2 -19138.15} C_VEL
LIN {X 0,Y 265.185,Z 892.289,A -85,B 0,C 180,E1 -19139.102,E2 -19139.102} C_VEL
LIN {X 0,Y 262.513,Z 902.203,A -85,B 0,C 180,E1 -19140.088,E2 -19140.088} C_VEL
LIN {X 0,Y 259.645,Z 911.897,A -85,B 0,C 180,E1 -19141.283,E2 -19141.283} C_VEL
LIN {X 0,Y 256.578,Z 921.286,A -85,B 0,C 180,E1 -19142.688,E2 -19142.688} C_VEL
LIN {X 0,Y 253.739,Z 929.438,A -85,B 0,C 180,E1 -19144.133,E2 -19144.133} C_VEL
LIN {X 0,Y 250.627,Z 938.092,A -85,B 0,C 180,E1 -19146.006,E2 -19146.006} C_VEL
LIN {X 0,Y 247.99,Z 945.448,A -85,B 0,C 180,E1 -19147.942,E2 -19147.942} C_VEL
LIN {X 0,Y 245.734,Z 951.8,A -85,B 0,C 180,E1 -19149.926,E2 -19149.926} C_VEL
LIN {X 0,Y 243.867,Z 957.317,A -85,B 0,C 180,E1 -19151.995,E2 -19151.995} C_VEL
LIN {X 0,Y 242.164,Z 963.325,A -85,B 0,C 180,E1 -19154.857,E2 -19154.857} C_VEL
LIN {X 0,Y 241.223,Z 967.472,A -85,B 0,C 180,E1 -19157.376,E2 -19157.376} C_VEL
LIN {X 0,Y 240.886,Z 970.645,A -85,B 0,C 180,E1 -19159.916,E2 -19159.916} C_VEL
LIN {X 0,Y 241.03,Z 973.178,A -85,B 0,C 180,E1 -19162.471,E2 -19162.471} C_VEL
LIN {X 0,Y 241.274,Z 976.016,A -85,B 0,C 180,E1 -19164.984,E2 -19164.984} C_VEL
LIN {X 0,Y 241.493,Z 977.346,A -85,B 0,C 180,E1 -19166.661,E2 -19166.661} C_VEL
LIN {X 0,Y 241.701,Z 978.245,A -85,B 0,C 180,E1 -19168.331,E2 -19168.331} C_VEL
LIN {X 0,Y 241.888,Z 978.7,A -85,B 0,C 180,E1 -19169.998,E2 -19169.998} C_VEL
LIN {X 0,Y 241.656,Z 978.634,A -85,B 0,C 180,E1 -19171.664,E2 -19171.664} C_VEL
LIN {X 0,Y 241.433,Z 978.156,A -85,B 0,C 180,E1 -19173.335,E2 -19173.335} C_VEL
LIN {X 0,Y 241.204,Z 977.265,A -85,B 0,C 180,E1 -19175.012,E2 -19175.012} C_VEL
LIN {X 0,Y 240.878,Z 975.391,A -85,B 0,C 180,E1 -19177.25,E2 -19177.25} C_VEL
LIN {X 0,Y 240.813,Z 971.964,A -85,B 0,C 180,E1 -19180.082,E2 -19180.082} C_VEL
LIN {X 0,Y 241.203,Z 967.816,A -85,B 0,C 180,E1 -19182.62,E2 -19182.62} C_VEL
LIN {X 0,Y 242.319,Z 961.598,A -85,B 0,C 180,E1 -19185.559,E2 -19185.559} C_VEL
LIN {X 0,Y 243.667,Z 955.44,A -85,B 0,C 180,E1 -19187.86,E2 -19187.86} C_VEL
LIN {X 0,Y 245.547,Z 948.128,A -85,B 0,C 180,E1 -19190.085,E2 -19190.085} C_VEL
LIN {X 0,Y 247.67,Z 940.084,A -85,B 0,C 180,E1 -19192.083,E2 -19192.083} C_VEL
LIN {X 0,Y 250.535,Z 929.267,A -85,B 0,C 180,E1 -19194.218,E2 -19194.218} C_VEL
LIN {X 0,Y 253.176,Z 918.34,A -85,B 0,C 180,E1 -19195.923,E2 -19195.923} C_VEL
LIN {X 0,Y 255.506,Z 907.798,A -85,B 0,C 180,E1 -19197.21,E2 -19197.21} C_VEL
LIN {X 0,Y 257.838,Z 895.222,A -85,B 0,C 180,E1 -19198.376,E2 -19198.376} C_VEL
LIN {X 0,Y 259.594,Z 882.002,A -85,B 0,C 180,E1 -19199.28,E2 -19199.28} C_VEL
LIN {X 0,Y 260.747,Z 869.265,A -85,B 0,C 180,E1 -19199.852,E2 -19199.852} C_VEL
LIN {X 0,Y 261.984,Z 836.503,A -85,B 0,C 180,E1 -19200.81,E2 -19200.81} C_VEL
LIN {X 0,Y 260.134,Z 810.611,A -85,B 0,C 180,E1 -19201.984,E2 -19201.984} C_VEL
LIN {X 0,Y 257.809,Z 787.598,A -85,B 0,C 180,E1 -19203.171,E2 -19203.171} C_VEL
LIN {X 0,Y 254.426,Z 765.459,A -85,B 0,C 180,E1 -19204.559,E2 -19204.559} C_VEL
LIN {X 0,Y 251.238,Z 757.532,A -85,B 0,C 180,E1 -19205.506,E2 -19205.506} C_VEL
LIN {X 0,Y 249.284,Z 748.076,A -85,B 0,C 180,E1 -19208.717,E2 -19208.717} C_VEL
LIN {X 0,Y 246.572,Z 737.535,A -85,B 0,C 180,E1 -19212.754,E2 -19212.754} C_VEL
LIN {X 0,Y 243.905,Z 728.603,A -85,B 0,C 180,E1 -19216.587,E2 -19216.587} C_VEL
LIN {X 0,Y 242.003,Z 722.418,A -85,B 0,C 180,E1 -19219.601,E2 -19219.601} C_VEL
LIN {X 0,Y 242.019,Z 722.316,A -85,B 0,C 180,E1 -19224.394,E2 -19224.394} C_VEL
LIN {X 0,Y 241.966,Z 722.34,A -85,B 0,C 180,E1 -19228.479,E2 -19228.479} C_VEL
LIN {X 0,Y 241.999,Z 722.335,A -85,B 0,C 180,E1 -19232.312,E2 -19232.312} C_VEL
LIN {X 0,Y 242.047,Z 722.33,A -85,B 0,C 180,E1 -19236.015,E2 -19236.015} C_VEL
LIN {X 0,Y 242.027,Z 722.33,A -85,B 0,C 180,E1 -19239.607,E2 -19239.607} C_VEL
LIN {X 0,Y 242.152,Z 722.312,A -85,B 0,C 180,E1 -19243.278,E2 -19243.278} C_VEL
LIN {X 0,Y 242.169,Z 722.318,A -85,B 0,C 180,E1 -19248.279,E2 -19248.279} C_VEL
LIN {X 0,Y 242.389,Z 722.279,A -85,B 0,C 180,E1 -19251.664,E2 -19251.664} C_VEL
LIN {X 0,Y 242.247,Z 722.299,A -85,B 0,C 180,E1 -19255.007,E2 -19255.007} C_VEL
LIN {X 0,Y 242.625,Z 722.262,A -85,B 0,C 180,E1 -19258.34,E2 -19258.34} C_VEL
LIN {X 0,Y 242.625,Z 722.259,A -85,B 0,C 180,E1 -19261.66,E2 -19261.66} C_VEL
LIN {X 0,Y 242.413,Z 722.289,A -85,B 0,C 180,E1 -19266.811,E2 -19266.811} C_VEL
LIN {X 0,Y 242.303,Z 722.301,A -85,B 0,C 180,E1 -19270.023,E2 -19270.023} C_VEL
LIN {X 0,Y 242.156,Z 722.316,A -85,B 0,C 180,E1 -19275.142,E2 -19275.142} C_VEL
LIN {X 0,Y 242.061,Z 722.328,A -85,B 0,C 180,E1 -19278.625,E2 -19278.625} C_VEL
LIN {X 0,Y 241.996,Z 722.323,A -85,B 0,C 180,E1 -19282.182,E2 -19282.182} C_VEL
LIN {X 0,Y 242.057,Z 722.331,A -85,B 0,C 180,E1 -19285.84,E2 -19285.84} C_VEL
LIN {X 0,Y 242.047,Z 722.559,A -85,B 0,C 180,E1 -19288.154,E2 -19288.154} C_VEL
LIN {X 0,Y 242.278,Z 723.51,A -85,B 0,C 180,E1 -19288.478,E2 -19288.478} C_VEL
LIN {X 0,Y 243.792,Z 726.208,A -85,B 0,C 180,E1 -19288.942,E2 -19288.942} C_VEL
LIN {X 0,Y 244.96,Z 727.604,A -85,B 0,C 180,E1 -19289.251,E2 -19289.251} C_VEL
LIN {X 0,Y 247.133,Z 730.978,A -85,B 0,C 180,E1 -19289.846,E2 -19289.846} C_VEL
LIN {X 0,Y 255.769,Z 745.034,A -85,B 0,C 180,E1 -19292.042,E2 -19292.042} C_VEL
LIN {X 0,Y 262.572,Z 757.974,A -85,B 0,C 180,E1 -19293.665,E2 -19293.665} C_VEL
LIN {X 0,Y 264.856,Z 762.867,A -85,B 0,C 180,E1 -19294.203,E2 -19294.203} C_VEL
LIN {X 0,Y 263.663,Z 800.628,A -85,B 0,C 180,E1 -19295.331,E2 -19295.331} C_VEL
LIN {X 0,Y 263.297,Z 814.969,A -85,B 0,C 180,E1 -19295.917,E2 -19295.917} C_VEL
LIN {X 0,Y 262.516,Z 827.417,A -85,B 0,C 180,E1 -19296.733,E2 -19296.733} C_VEL
LIN {X 0,Y 261.263,Z 839.371,A -85,B 0,C 180,E1 -19297.802,E2 -19297.802} C_VEL
LIN {X 0,Y 259.52,Z 851.153,A -85,B 0,C 180,E1 -19299.182,E2 -19299.182} C_VEL
LIN {X 0,Y 257.584,Z 861.57,A -85,B 0,C 180,E1 -19300.751,E2 -19300.751} C_VEL
LIN {X 0,Y 255.4,Z 871.421,A -85,B 0,C 180,E1 -19302.604,E2 -19302.604} C_VEL
LIN {X 0,Y 253.39,Z 879.278,A -85,B 0,C 180,E1 -19304.426,E2 -19304.426} C_VEL
LIN {X 0,Y 251.177,Z 887.139,A -85,B 0,C 180,E1 -19306.677,E2 -19306.677} C_VEL
LIN {X 0,Y 249.172,Z 893.619,A -85,B 0,C 180,E1 -19309.025,E2 -19309.025} C_VEL
LIN {X 0,Y 247.479,Z 898.684,A -85,B 0,C 180,E1 -19311.339,E2 -19311.339} C_VEL
LIN {X 0,Y 245.716,Z 903.311,A -85,B 0,C 180,E1 -19314.105,E2 -19314.105} C_VEL
LIN {X 0,Y 244.467,Z 906.585,A -85,B 0,C 180,E1 -19316.895,E2 -19316.895} C_VEL
LIN {X 0,Y 243.493,Z 908.789,A -85,B 0,C 180,E1 -19319.987,E2 -19319.987} C_VEL
LIN {X 0,Y 242.987,Z 909.535,A -85,B 0,C 180,E1 -19322.437,E2 -19322.437} C_VEL
LIN {X 0,Y 242.788,Z 909.515,A -85,B 0,C 180,E1 -19324.268,E2 -19324.268} C_VEL
LIN {X 0,Y 242.709,Z 909.044,A -85,B 0,C 180,E1 -19326.087,E2 -19326.087} C_VEL
LIN {X 0,Y 242.781,Z 908.129,A -85,B 0,C 180,E1 -19327.897,E2 -19327.897} C_VEL
LIN {X 0,Y 243.028,Z 906.698,A -85,B 0,C 180,E1 -19329.698,E2 -19329.698} C_VEL
LIN {X 0,Y 243.586,Z 903.924,A -85,B 0,C 180,E1 -19332.2,E2 -19332.2} C_VEL
LIN {X 0,Y 244.549,Z 899.565,A -85,B 0,C 180,E1 -19335.013,E2 -19335.013} C_VEL
LIN {X 0,Y 245.758,Z 894.061,A -85,B 0,C 180,E1 -19337.686,E2 -19337.686} C_VEL
LIN {X 0,Y 247.168,Z 887.471,A -85,B 0,C 180,E1 -19340.18,E2 -19340.18} C_VEL
LIN {X 0,Y 248.97,Z 878.704,A -85,B 0,C 180,E1 -19342.789,E2 -19342.789} C_VEL
LIN {X 0,Y 250.582,Z 870.395,A -85,B 0,C 180,E1 -19344.773,E2 -19344.773} C_VEL
LIN {X 0,Y 252.226,Z 860.971,A -85,B 0,C 180,E1 -19346.608,E2 -19346.608} C_VEL
LIN {X 0,Y 253.746,Z 850.809,A -85,B 0,C 180,E1 -19348.204,E2 -19348.204} C_VEL
LIN {X 0,Y 255.164,Z 839.582,A -85,B 0,C 180,E1 -19349.608,E2 -19349.608} C_VEL
LIN {X 0,Y 256.313,Z 827.41,A -85,B 0,C 180,E1 -19350.788,E2 -19350.788} C_VEL
LIN {X 0,Y 257.052,Z 814.353,A -85,B 0,C 180,E1 -19351.705,E2 -19351.705} C_VEL
LIN {X 0,Y 257.413,Z 800.82,A -85,B 0,C 180,E1 -19352.319,E2 -19352.319} C_VEL
LIN {X 0,Y 258.336,Z 756.459,A -85,B 0,C 180,E1 -19353.634,E2 -19353.634} C_VEL
LIN {X 0,Y 251.353,Z 740.684,A -85,B 0,C 180,E1 -19354.945,E2 -19354.945} C_VEL
LIN {X 0,Y 242.587,Z 723.267,A -85,B 0,C 180,E1 -19356.657,E2 -19356.657} C_VEL
LIN {X 0,Y 242.378,Z 722.368,A -85,B 0,C 180,E1 -19357.029,E2 -19357.029} C_VEL
LIN {X 0,Y 242.265,Z 722.299,A -85,B 0,C 180,E1 -19360.026,E2 -19360.026} C_VEL
LIN {X 0,Y 242.127,Z 722.31,A -85,B 0,C 180,E1 -19365.146,E2 -19365.146} C_VEL
LIN {X 0,Y 242.027,Z 722.325,A -85,B 0,C 180,E1 -19368.63,E2 -19368.63} C_VEL
LIN {X 0,Y 241.979,Z 722.341,A -85,B 0,C 180,E1 -19372.186,E2 -19372.186} C_VEL
LIN {X 0,Y 241.993,Z 722.316,A -85,B 0,C 180,E1 -19375.828,E2 -19375.828} C_VEL
LIN {X 0,Y 241.969,Z 722.343,A -85,B 0,C 180,E1 -19379.591,E2 -19379.591} C_VEL
LIN {X 0,Y 241.985,Z 722.312,A -85,B 0,C 180,E1 -19383.495,E2 -19383.495} C_VEL
LIN {X 0,Y 241.991,Z 722.327,A -85,B 0,C 180,E1 -19387.584,E2 -19387.584} C_VEL
LIN {X 0,Y 241.914,Z 722.352,A -85,B 0,C 180,E1 -19391.93,E2 -19391.93} C_VEL
LIN {X 0,Y 241.908,Z 722.352,A -85,B 0,C 180,E1 -19396.581,E2 -19396.581} C_VEL
LIN {X 0,Y 241.991,Z 722.518,A -85,B 0,C 180,E1 -19399.949,E2 -19399.949} C_VEL
LIN {X 0,Y 242.217,Z 723.53,A -85,B 0,C 180,E1 -19400.22,E2 -19400.22} C_VEL
LIN {X 0,Y 251.521,Z 750.109,A -85,B 0,C 180,E1 -19401.983,E2 -19401.983} C_VEL
LIN {X 0,Y 249.888,Z 801.009,A -85,B 0,C 180,E1 -19404.015,E2 -19404.015} C_VEL
LIN {X 0,Y 249.437,Z 813.042,A -85,B 0,C 180,E1 -19404.727,E2 -19404.727} C_VEL
LIN {X 0,Y 248.802,Z 824.04,A -85,B 0,C 180,E1 -19405.601,E2 -19405.601} C_VEL
LIN {X 0,Y 248.173,Z 832.963,A -85,B 0,C 180,E1 -19406.48,E2 -19406.48} C_VEL
LIN {X 0,Y 247.316,Z 843.627,A -85,B 0,C 180,E1 -19407.777,E2 -19407.777} C_VEL
LIN {X 0,Y 246.469,Z 852.767,A -85,B 0,C 180,E1 -19409.118,E2 -19409.118} C_VEL
LIN {X 0,Y 245.645,Z 861.594,A -85,B 0,C 180,E1 -19410.662,E2 -19410.662} C_VEL
LIN {X 0,Y 244.902,Z 869.114,A -85,B 0,C 180,E1 -19412.203,E2 -19412.203} C_VEL
LIN {X 0,Y 244.052,Z 876.569,A -85,B 0,C 180,E1 -19413.997,E2 -19413.997} C_VEL
LIN {X 0,Y 243.377,Z 884.036,A -85,B 0,C 180,E1 -19416.154,E2 -19416.154} C_VEL
LIN {X 0,Y 242.822,Z 890.345,A -85,B 0,C 180,E1 -19418.344,E2 -19418.344} C_VEL
LIN {X 0,Y 242.462,Z 895.55,A -85,B 0,C 180,E1 -19420.528,E2 -19420.528} C_VEL
LIN {X 0,Y 242.288,Z 899.09,A -85,B 0,C 180,E1 -19422.267,E2 -19422.267} C_VEL
LIN {X 0,Y 242.304,Z 903.193,A -85,B 0,C 180,E1 -19424.868,E2 -19424.868} C_VEL
LIN {X 0,Y 242.442,Z 905.316,A -85,B 0,C 180,E1 -19426.59,E2 -19426.59} C_VEL
LIN {X 0,Y 243.165,Z 908.13,A -85,B 0,C 180,E1 -19430.013,E2 -19430.013} C_VEL
LIN {X 0,Y 243.683,Z 908.872,A -85,B 0,C 180,E1 -19431.708,E2 -19431.708} C_VEL
LIN {X 0,Y 244.384,Z 909.161,A -85,B 0,C 180,E1 -19433.394,E2 -19433.394} C_VEL
LIN {X 0,Y 246.343,Z 908.304,A -85,B 0,C 180,E1 -19436.924,E2 -19436.924} C_VEL
LIN {X 0,Y 248.51,Z 905.838,A -85,B 0,C 180,E1 -19440,E2 -19440} C_VEL
LIN {X 0,Y 249.819,Z 904.044,A -85,B 0,C 180,E1 -19441.565,E2 -19441.565} C_VEL
LIN {X 0,Y 250.399,Z 902.546,A -85,B 0,C 180,E1 -19442.869,E2 -19442.869} C_VEL
LIN {X 0,Y 249.878,Z 899.824,A -85,B 0,C 180,E1 -19445.052,E2 -19445.052} C_VEL
LIN {X 0,Y 249.603,Z 896.394,A -85,B 0,C 180,E1 -19447.176,E2 -19447.176} C_VEL
LIN {X 0,Y 250.533,Z 893.666,A -85,B 0,C 180,E1 -19448.36,E2 -19448.36} C_VEL
LIN {X 0,Y 252.81,Z 888.871,A -85,B 0,C 180,E1 -19450.006,E2 -19450.006} C_VEL
LIN {X 0,Y 255.744,Z 882.167,A -85,B 0,C 180,E1 -19451.894,E2 -19451.894} C_VEL
LIN {X 0,Y 258.225,Z 875.903,A -85,B 0,C 180,E1 -19453.376,E2 -19453.376} C_VEL
LIN {X 0,Y 261.098,Z 867.579,A -85,B 0,C 180,E1 -19455.015,E2 -19455.015} C_VEL
LIN {X 0,Y 263.422,Z 859.898,A -85,B 0,C 180,E1 -19456.269,E2 -19456.269} C_VEL
LIN {X 0,Y 265.785,Z 850.87,A -85,B 0,C 180,E1 -19457.504,E2 -19457.504} C_VEL
LIN {X 0,Y 267.831,Z 841.64,A -85,B 0,C 180,E1 -19458.552,E2 -19458.552} C_VEL
LIN {X 0,Y 269.447,Z 832.416,A -85,B 0,C 180,E1 -19459.424,E2 -19459.424} C_VEL
LIN {X 0,Y 270.887,Z 821.894,A -85,B 0,C 180,E1 -19460.205,E2 -19460.205} C_VEL
LIN {X 0,Y 272.739,Z 803.458,A -85,B 0,C 180,E1 -19461.218,E2 -19461.218} C_VEL
LIN {X 0,Y 275.688,Z 777.483,A -85,B 0,C 180,E1 -19462.403,E2 -19462.403} C_VEL
LIN {X 0,Y 272.057,Z 770.348,A -85,B 0,C 180,E1 -19464.501,E2 -19464.501} C_VEL
LIN {X 0,Y 269.109,Z 765.317,A -85,B 0,C 180,E1 -19466.488,E2 -19466.488} C_VEL
LIN {X 0,Y 267.17,Z 762.045,A -85,B 0,C 180,E1 -19468.078,E2 -19468.078} C_VEL
LIN {X 0,Y 265.248,Z 758.782,A -85,B 0,C 180,E1 -19470.026,E2 -19470.026} C_VEL
LIN {X 0,Y 264.742,Z 758.074,A -85,B 0,C 180,E1 -19470.609,E2 -19470.609} C_VEL
LIN {X 0,Y 262.705,Z 755.249,A -85,B 0,C 180,E1 -19473.967,E2 -19473.967} C_VEL
LIN {X 0,Y 262.52,Z 754.704,A -85,B 0,C 180,E1 -19474.664,E2 -19474.664} C_VEL
LIN {X 0,Y 261.977,Z 754.965,A -85,B 0,C 180,E1 -19477.336,E2 -19477.336} C_VEL
LIN {X 0,Y 262.814,Z 757.039,A -85,B 0,C 180,E1 -19481.148,E2 -19481.148} C_VEL
LIN {X 0,Y 263.73,Z 759.057,A -85,B 0,C 180,E1 -19482.867,E2 -19482.867} C_VEL
LIN {X 0,Y 265.69,Z 762.346,A -85,B 0,C 180,E1 -19485.226,E2 -19485.226} C_VEL
LIN {X 0,Y 266.562,Z 764.478,A -85,B 0,C 180,E1 -19486.183,E2 -19486.183} C_VEL
LIN {X 0,Y 268.14,Z 772.859,A -85,B 0,C 180,E1 -19488.219,E2 -19488.219} C_VEL
LIN {X 0,Y 270.238,Z 782.712,A -85,B 0,C 180,E1 -19490.295,E2 -19490.295} C_VEL
LIN {X 0,Y 270.268,Z 802.144,A -85,B 0,C 180,E1 -19492.164,E2 -19492.164} C_VEL
LIN {X 0,Y 270.012,Z 822.828,A -85,B 0,C 180,E1 -19493.836,E2 -19493.836} C_VEL
LIN {X 0,Y 268.985,Z 843.858,A -85,B 0,C 180,E1 -19495.146,E2 -19495.146} C_VEL
LIN {X 0,Y 266.311,Z 864.883,A -85,B 0,C 180,E1 -19496.08,E2 -19496.08} C_VEL
LIN {X 0,Y 263.432,Z 879.359,A -85,B 0,C 180,E1 -19496.956,E2 -19496.956} C_VEL
LIN {X 0,Y 260.67,Z 890.361,A -85,B 0,C 180,E1 -19497.824,E2 -19497.824} C_VEL
LIN {X 0,Y 257.87,Z 900.239,A -85,B 0,C 180,E1 -19498.811,E2 -19498.811} C_VEL
LIN {X 0,Y 254.363,Z 911.16,A -85,B 0,C 180,E1 -19500.174,E2 -19500.174} C_VEL
LIN {X 0,Y 251.135,Z 920.462,A -85,B 0,C 180,E1 -19501.59,E2 -19501.59} C_VEL
LIN {X 0,Y 248.089,Z 928.479,A -85,B 0,C 180,E1 -19503.045,E2 -19503.045} C_VEL
LIN {X 0,Y 244.769,Z 937.001,A -85,B 0,C 180,E1 -19504.941,E2 -19504.941} C_VEL
LIN {X 0,Y 241.952,Z 944.32,A -85,B 0,C 180,E1 -19506.91,E2 -19506.91} C_VEL
LIN {X 0,Y 239.485,Z 950.591,A -85,B 0,C 180,E1 -19508.929,E2 -19508.929} C_VEL
LIN {X 0,Y 237.518,Z 955.968,A -85,B 0,C 180,E1 -19511.003,E2 -19511.003} C_VEL
LIN {X 0,Y 236.197,Z 959.627,A -85,B 0,C 180,E1 -19512.687,E2 -19512.687} C_VEL
LIN {X 0,Y 234.538,Z 965.607,A -85,B 0,C 180,E1 -19516.127,E2 -19516.127} C_VEL
LIN {X 0,Y 233.833,Z 969.745,A -85,B 0,C 180,E1 -19519.608,E2 -19519.608} C_VEL
LIN {X 0,Y 233.973,Z 972.252,A -85,B 0,C 180,E1 -19522.412,E2 -19522.412} C_VEL
LIN {X 0,Y 234.209,Z 974.914,A -85,B 0,C 180,E1 -19524.833,E2 -19524.833} C_VEL
LIN {X 0,Y 234.434,Z 976.266,A -85,B 0,C 180,E1 -19526.56,E2 -19526.56} C_VEL
LIN {X 0,Y 234.655,Z 977.185,A -85,B 0,C 180,E1 -19528.281,E2 -19528.281} C_VEL
LIN {X 0,Y 234.855,Z 977.672,A -85,B 0,C 180,E1 -19529.997,E2 -19529.997} C_VEL
LIN {X 0,Y 234.607,Z 977.626,A -85,B 0,C 180,E1 -19531.714,E2 -19531.714} C_VEL
LIN {X 0,Y 234.377,Z 977.162,A -85,B 0,C 180,E1 -19533.436,E2 -19533.436} C_VEL
LIN {X 0,Y 234.117,Z 976.281,A -85,B 0,C 180,E1 -19535.164,E2 -19535.164} C_VEL
LIN {X 0,Y 233.816,Z 974.612,A -85,B 0,C 180,E1 -19537.293,E2 -19537.293} C_VEL
LIN {X 0,Y 233.747,Z 971.044,A -85,B 0,C 180,E1 -19540.39,E2 -19540.39} C_VEL
LIN {X 0,Y 234.217,Z 966.947,A -85,B 0,C 180,E1 -19543.003,E2 -19543.003} C_VEL
LIN {X 0,Y 235.18,Z 961.75,A -85,B 0,C 180,E1 -19545.599,E2 -19545.599} C_VEL
LIN {X 0,Y 236.497,Z 955.929,A -85,B 0,C 180,E1 -19547.943,E2 -19547.943} C_VEL
LIN {X 0,Y 238.464,Z 948.847,A -85,B 0,C 180,E1 -19550.258,E2 -19550.258} C_VEL
LIN {X 0,Y 241.103,Z 939.477,A -85,B 0,C 180,E1 -19552.717,E2 -19552.717} C_VEL
LIN {X 0,Y 244.053,Z 928.768,A -85,B 0,C 180,E1 -19554.905,E2 -19554.905} C_VEL
LIN {X 0,Y 246.822,Z 917.956,A -85,B 0,C 180,E1 -19556.642,E2 -19556.642} C_VEL
LIN {X 0,Y 249.6,Z 905.92,A -85,B 0,C 180,E1 -19558.137,E2 -19558.137} C_VEL
LIN {X 0,Y 252.003,Z 893.148,A -85,B 0,C 180,E1 -19559.324,E2 -19559.324} C_VEL
LIN {X 0,Y 253.73,Z 880.836,A -85,B 0,C 180,E1 -19560.163,E2 -19560.163} C_VEL
LIN {X 0,Y 254.889,Z 867.851,A -85,B 0,C 180,E1 -19560.759,E2 -19560.759} C_VEL
LIN {X 0,Y 256.123,Z 837.664,A -85,B 0,C 180,E1 -19561.658,E2 -19561.658} C_VEL
LIN {X 0,Y 254.358,Z 811.648,A -85,B 0,C 180,E1 -19562.871,E2 -19562.871} C_VEL
LIN {X 0,Y 252.153,Z 789.055,A -85,B 0,C 180,E1 -19564.072,E2 -19564.072} C_VEL
LIN {X 0,Y 249.192,Z 768.576,A -85,B 0,C 180,E1 -19565.396,E2 -19565.396} C_VEL
LIN {X 0,Y 245.259,Z 759.579,A -85,B 0,C 180,E1 -19566.51,E2 -19566.51} C_VEL
LIN {X 0,Y 243.878,Z 755.987,A -85,B 0,C 180,E1 -19567.029,E2 -19567.029} C_VEL
LIN {X 0,Y 241.979,Z 747.427,A -85,B 0,C 180,E1 -19570.131,E2 -19570.131} C_VEL
LIN {X 0,Y 239.392,Z 737.906,A -85,B 0,C 180,E1 -19574.008,E2 -19574.008} C_VEL
LIN {X 0,Y 237.402,Z 731.081,A -85,B 0,C 180,E1 -19577.087,E2 -19577.087} C_VEL
LIN {X 0,Y 234.939,Z 723.301,A -85,B 0,C 180,E1 -19581.083,E2 -19581.083} C_VEL
LIN {X 0,Y 234.951,Z 723.197,A -85,B 0,C 180,E1 -19585.366,E2 -19585.366} C_VEL
LIN {X 0,Y 234.96,Z 723.219,A -85,B 0,C 180,E1 -19590.156,E2 -19590.156} C_VEL
LIN {X 0,Y 234.984,Z 723.214,A -85,B 0,C 180,E1 -19593.793,E2 -19593.793} C_VEL
LIN {X 0,Y 235.001,Z 723.202,A -85,B 0,C 180,E1 -19598.969,E2 -19598.969} C_VEL
LIN {X 0,Y 235.085,Z 723.191,A -85,B 0,C 180,E1 -19603.059,E2 -19603.059} C_VEL
LIN {X 0,Y 235.103,Z 723.194,A -85,B 0,C 180,E1 -19607.922,E2 -19607.922} C_VEL
LIN {X 0,Y 235.32,Z 723.158,A -85,B 0,C 180,E1 -19611.412,E2 -19611.412} C_VEL
LIN {X 0,Y 235.381,Z 723.165,A -85,B 0,C 180,E1 -19613.141,E2 -19613.141} C_VEL
LIN {X 0,Y 235.585,Z 723.139,A -85,B 0,C 180,E1 -19618.291,E2 -19618.291} C_VEL
LIN {X 0,Y 235.585,Z 723.136,A -85,B 0,C 180,E1 -19621.71,E2 -19621.71} C_VEL
LIN {X 0,Y 235.393,Z 723.164,A -85,B 0,C 180,E1 -19626.859,E2 -19626.859} C_VEL
LIN {X 0,Y 235.227,Z 723.184,A -85,B 0,C 180,E1 -19630.327,E2 -19630.327} C_VEL
LIN {X 0,Y 235.104,Z 723.192,A -85,B 0,C 180,E1 -19635.607,E2 -19635.607} C_VEL
LIN {X 0,Y 234.997,Z 723.206,A -85,B 0,C 180,E1 -19639.207,E2 -19639.207} C_VEL
LIN {X 0,Y 234.943,Z 723.195,A -85,B 0,C 180,E1 -19642.885,E2 -19642.885} C_VEL
LIN {X 0,Y 234.99,Z 723.436,A -85,B 0,C 180,E1 -19646.543,E2 -19646.543} C_VEL
LIN {X 0,Y 235.265,Z 724.531,A -85,B 0,C 180,E1 -19646.922,E2 -19646.922} C_VEL
LIN {X 0,Y 236.715,Z 727.076,A -85,B 0,C 180,E1 -19647.401,E2 -19647.401} C_VEL
LIN {X 0,Y 238.011,Z 728.455,A -85,B 0,C 180,E1 -19647.763,E2 -19647.763} C_VEL
LIN {X 0,Y 240.193,Z 731.875,A -85,B 0,C 180,E1 -19648.407,E2 -19648.407} C_VEL
LIN {X 0,Y 246.148,Z 741.214,A -85,B 0,C 180,E1 -19650.059,E2 -19650.059} C_VEL
LIN {X 0,Y 251.822,Z 750.833,A -85,B 0,C 180,E1 -19651.539,E2 -19651.539} C_VEL
LIN {X 0,Y 257.723,Z 762.259,A -85,B 0,C 180,E1 -19653.015,E2 -19653.015} C_VEL
LIN {X 0,Y 259.061,Z 765.124,A -85,B 0,C 180,E1 -19653.343,E2 -19653.343} C_VEL
LIN {X 0,Y 257.859,Z 801.881,A -85,B 0,C 180,E1 -19654.47,E2 -19654.47} C_VEL
LIN {X 0,Y 257.471,Z 815.491,A -85,B 0,C 180,E1 -19655.031,E2 -19655.031} C_VEL
LIN {X 0,Y 256.741,Z 827.395,A -85,B 0,C 180,E1 -19655.816,E2 -19655.816} C_VEL
LIN {X 0,Y 255.4,Z 839.55,A -85,B 0,C 180,E1 -19656.9,E2 -19656.9} C_VEL
LIN {X 0,Y 253.671,Z 850.908,A -85,B 0,C 180,E1 -19658.226,E2 -19658.226} C_VEL
LIN {X 0,Y 251.539,Z 862.054,A -85,B 0,C 180,E1 -19659.906,E2 -19659.906} C_VEL
LIN {X 0,Y 249.1,Z 872.574,A -85,B 0,C 180,E1 -19661.92,E2 -19661.92} C_VEL
LIN {X 0,Y 246.741,Z 881.311,A -85,B 0,C 180,E1 -19664.015,E2 -19664.015} C_VEL
LIN {X 0,Y 244.39,Z 889.054,A -85,B 0,C 180,E1 -19666.36,E2 -19666.36} C_VEL
LIN {X 0,Y 242.162,Z 895.866,A -85,B 0,C 180,E1 -19668.989,E2 -19668.989} C_VEL
LIN {X 0,Y 239.94,Z 901.87,A -85,B 0,C 180,E1 -19672.044,E2 -19672.044} C_VEL
LIN {X 0,Y 238.3,Z 905.891,A -85,B 0,C 180,E1 -19674.898,E2 -19674.898} C_VEL
LIN {X 0,Y 237.14,Z 908.613,A -85,B 0,C 180,E1 -19677.764,E2 -19677.764} C_VEL
LIN {X 0,Y 236.547,Z 909.789,A -85,B 0,C 180,E1 -19679.666,E2 -19679.666} C_VEL
LIN {X 0,Y 236.128,Z 910.416,A -85,B 0,C 180,E1 -19681.565,E2 -19681.565} C_VEL
LIN {X 0,Y 235.838,Z 910.598,A -85,B 0,C 180,E1 -19683.452,E2 -19683.452} C_VEL
LIN {X 0,Y 235.693,Z 910.301,A -85,B 0,C 180,E1 -19685.329,E2 -19685.329} C_VEL
LIN {X 0,Y 235.726,Z 909.33,A -85,B 0,C 180,E1 -19687.556,E2 -19687.556} C_VEL
LIN {X 0,Y 235.883,Z 908.307,A -85,B 0,C 180,E1 -19689.054,E2 -19689.054} C_VEL
LIN {X 0,Y 236.484,Z 905.352,A -85,B 0,C 180,E1 -19691.991,E2 -19691.991} C_VEL
LIN {X 0,Y 237.342,Z 901.703,A -85,B 0,C 180,E1 -19694.547,E2 -19694.547} C_VEL
LIN {X 0,Y 238.565,Z 896.159,A -85,B 0,C 180,E1 -19697.456,E2 -19697.456} C_VEL
LIN {X 0,Y 240.189,Z 889.054,A -85,B 0,C 180,E1 -19700.317,E2 -19700.317} C_VEL
LIN {X 0,Y 241.809,Z 881.565,A -85,B 0,C 180,E1 -19702.682,E2 -19702.682} C_VEL
LIN {X 0,Y 243.673,Z 872.253,A -85,B 0,C 180,E1 -19705.039,E2 -19705.039} C_VEL
LIN {X 0,Y 245.488,Z 862.292,A -85,B 0,C 180,E1 -19707.06,E2 -19707.06} C_VEL
LIN {X 0,Y 247.167,Z 851.61,A -85,B 0,C 180,E1 -19708.78,E2 -19708.78} C_VEL
LIN {X 0,Y 248.636,Z 840.452,A -85,B 0,C 180,E1 -19710.205,E2 -19710.205} C_VEL
LIN {X 0,Y 249.84,Z 828.249,A -85,B 0,C 180,E1 -19711.413,E2 -19711.413} C_VEL
LIN {X 0,Y 250.61,Z 815.285,A -85,B 0,C 180,E1 -19712.342,E2 -19712.342} C_VEL
LIN {X 0,Y 250.997,Z 801.382,A -85,B 0,C 180,E1 -19712.985,E2 -19712.985} C_VEL
LIN {X 0,Y 251.901,Z 758.142,A -85,B 0,C 180,E1 -19714.304,E2 -19714.304} C_VEL
LIN {X 0,Y 244.895,Z 742.639,A -85,B 0,C 180,E1 -19715.654,E2 -19715.654} C_VEL
LIN {X 0,Y 235.514,Z 724.162,A -85,B 0,C 180,E1 -19717.558,E2 -19717.558} C_VEL
LIN {X 0,Y 235.33,Z 723.24,A -85,B 0,C 180,E1 -19717.942,E2 -19717.942} C_VEL
LIN {X 0,Y 235.213,Z 723.175,A -85,B 0,C 180,E1 -19720.33,E2 -19720.33} C_VEL
LIN {X 0,Y 235.076,Z 723.19,A -85,B 0,C 180,E1 -19725.612,E2 -19725.612} C_VEL
LIN {X 0,Y 234.967,Z 723.198,A -85,B 0,C 180,E1 -19729.212,E2 -19729.212} C_VEL
LIN {X 0,Y 234.923,Z 723.224,A -85,B 0,C 180,E1 -19732.889,E2 -19732.889} C_VEL
LIN {X 0,Y 234.911,Z 723.195,A -85,B 0,C 180,E1 -19736.667,E2 -19736.667} C_VEL
LIN {X 0,Y 234.901,Z 723.225,A -85,B 0,C 180,E1 -19740.575,E2 -19740.575} C_VEL
LIN {X 0,Y 234.947,Z 723.193,A -85,B 0,C 180,E1 -19743.115,E2 -19743.115} C_VEL
LIN {X 0,Y 234.922,Z 723.196,A -85,B 0,C 180,E1 -19746.753,E2 -19746.753} C_VEL
LIN {X 0,Y 234.919,Z 723.22,A -85,B 0,C 180,E1 -19748.937,E2 -19748.937} C_VEL
LIN {X 0,Y 234.859,Z 723.232,A -85,B 0,C 180,E1 -19753.496,E2 -19753.496} C_VEL
LIN {X 0,Y 234.861,Z 723.23,A -85,B 0,C 180,E1 -19756.507,E2 -19756.507} C_VEL
LIN {X 0,Y 234.92,Z 723.395,A -85,B 0,C 180,E1 -19759.483,E2 -19759.483} C_VEL
LIN {X 0,Y 235.133,Z 724.305,A -85,B 0,C 180,E1 -19759.756,E2 -19759.756} C_VEL
LIN {X 0,Y 244.63,Z 751.551,A -85,B 0,C 180,E1 -19761.623,E2 -19761.623} C_VEL
LIN {X 0,Y 242.949,Z 801.763,A -85,B 0,C 180,E1 -19763.692,E2 -19763.692} C_VEL
LIN {X 0,Y 242.482,Z 814.32,A -85,B 0,C 180,E1 -19764.464,E2 -19764.464} C_VEL
LIN {X 0,Y 241.787,Z 825.052,A -85,B 0,C 180,E1 -19765.345,E2 -19765.345} C_VEL
LIN {X 0,Y 241.075,Z 834.907,A -85,B 0,C 180,E1 -19766.364,E2 -19766.364} C_VEL
LIN {X 0,Y 240.333,Z 843.965,A -85,B 0,C 180,E1 -19767.497,E2 -19767.497} C_VEL
LIN {X 0,Y 239.351,Z 854.375,A -85,B 0,C 180,E1 -19769.079,E2 -19769.079} C_VEL
LIN {X 0,Y 238.508,Z 863.087,A -85,B 0,C 180,E1 -19770.667,E2 -19770.667} C_VEL
LIN {X 0,Y 237.702,Z 870.761,A -85,B 0,C 180,E1 -19772.306,E2 -19772.306} C_VEL
LIN {X 0,Y 236.897,Z 877.777,A -85,B 0,C 180,E1 -19774.05,E2 -19774.05} C_VEL
LIN {X 0,Y 236.371,Z 884.05,A -85,B 0,C 180,E1 -19775.868,E2 -19775.868} C_VEL
LIN {X 0,Y 235.756,Z 890.808,A -85,B 0,C 180,E1 -19778.223,E2 -19778.223} C_VEL
LIN {X 0,Y 235.474,Z 895.019,A -85,B 0,C 180,E1 -19779.926,E2 -19779.926} C_VEL
LIN {X 0,Y 235.211,Z 900.958,A -85,B 0,C 180,E1 -19782.976,E2 -19782.976} C_VEL
LIN {X 0,Y 235.271,Z 904.453,A -85,B 0,C 180,E1 -19785.291,E2 -19785.291} C_VEL
LIN {X 0,Y 235.595,Z 907.41,A -85,B 0,C 180,E1 -19787.947,E2 -19787.947} C_VEL
LIN {X 0,Y 236.035,Z 908.858,A -85,B 0,C 180,E1 -19789.708,E2 -19789.708} C_VEL
LIN {X 0,Y 236.555,Z 909.805,A -85,B 0,C 180,E1 -19791.457,E2 -19791.457} C_VEL
LIN {X 0,Y 237.273,Z 910.29,A -85,B 0,C 180,E1 -19793.195,E2 -19793.195} C_VEL
LIN {X 0,Y 238.112,Z 910.363,A -85,B 0,C 180,E1 -19794.92,E2 -19794.92} C_VEL
LIN {X 0,Y 240.23,Z 909.122,A -85,B 0,C 180,E1 -19798.323,E2 -19798.323} C_VEL
LIN {X 0,Y 241.529,Z 907.937,A -85,B 0,C 180,E1 -19800,E2 -19800} C_VEL
LIN {X 0,Y 243.684,Z 905.233,A -85,B 0,C 180,E1 -19802.479,E2 -19802.479} C_VEL
LIN {X 0,Y 246.232,Z 901.426,A -85,B 0,C 180,E1 -19804.912,E2 -19804.912} C_VEL
LIN {X 0,Y 249.639,Z 895.419,A -85,B 0,C 180,E1 -19807.685,E2 -19807.685} C_VEL
LIN {X 0,Y 250.533,Z 893.666,A -85,B 0,C 180,E1 -19808.36,E2 -19808.36} C_VEL
LIN {X 0,Y 251.553,Z 890.858,A -85,B 0,C 180,E1 -19809.524,E2 -19809.524} C_VEL
LIN {X 0,Y 251.794,Z 886.338,A -85,B 0,C 180,E1 -19811.538,E2 -19811.538} C_VEL
LIN {X 0,Y 252.098,Z 881.241,A -85,B 0,C 180,E1 -19813.457,E2 -19813.457} C_VEL
LIN {X 0,Y 253.155,Z 877.438,A -85,B 0,C 180,E1 -19814.448,E2 -19814.448} C_VEL
LIN {X 0,Y 256.242,Z 869.103,A -85,B 0,C 180,E1 -19816.123,E2 -19816.123} C_VEL
LIN {X 0,Y 258.732,Z 861.549,A -85,B 0,C 180,E1 -19817.385,E2 -19817.385} C_VEL
LIN {X 0,Y 261.251,Z 852.62,A -85,B 0,C 180,E1 -19818.63,E2 -19818.63} C_VEL
LIN {X 0,Y 263.683,Z 842.237,A -85,B 0,C 180,E1 -19819.816,E2 -19819.816} C_VEL
LIN {X 0,Y 265.65,Z 831.719,A -85,B 0,C 180,E1 -19820.791,E2 -19820.791} C_VEL
LIN {X 0,Y 267.36,Z 819.583,A -85,B 0,C 180,E1 -19821.649,E2 -19821.649} C_VEL
LIN {X 0,Y 269.885,Z 796.334,A -85,B 0,C 180,E1 -19822.844,E2 -19822.844} C_VEL
LIN {X 0,Y 271.745,Z 781.202,A -85,B 0,C 180,E1 -19823.562,E2 -19823.562} C_VEL
LIN {X 0,Y 269.09,Z 775.718,A -85,B 0,C 180,E1 -19825.29,E2 -19825.29} C_VEL
LIN {X 0,Y 266.53,Z 771.191,A -85,B 0,C 180,E1 -19827.186,E2 -19827.186} C_VEL
LIN {X 0,Y 265.018,Z 768.538,A -85,B 0,C 180,E1 -19828.512,E2 -19828.512} C_VEL
LIN {X 0,Y 263.127,Z 765.002,A -85,B 0,C 180,E1 -19830.657,E2 -19830.657} C_VEL
LIN {X 0,Y 261.212,Z 762.463,A -85,B 0,C 180,E1 -19833.752,E2 -19833.752} C_VEL
LIN {X 0,Y 260.936,Z 761.626,A -85,B 0,C 180,E1 -19834.76,E2 -19834.76} C_VEL
LIN {X 0,Y 260.443,Z 761.871,A -85,B 0,C 180,E1 -19837.255,E2 -19837.255} C_VEL
LIN {X 0,Y 261.19,Z 763.955,A -85,B 0,C 180,E1 -19841.009,E2 -19841.009} C_VEL
LIN {X 0,Y 261.915,Z 765.723,A -85,B 0,C 180,E1 -19842.522,E2 -19842.522} C_VEL
LIN {X 0,Y 263.704,Z 769.002,A -85,B 0,C 180,E1 -19844.861,E2 -19844.861} C_VEL
LIN {X 0,Y 264.223,Z 770.502,A -85,B 0,C 180,E1 -19845.511,E2 -19845.511} C_VEL
LIN {X 0,Y 265.585,Z 779.201,A -85,B 0,C 180,E1 -19847.636,E2 -19847.636} C_VEL
LIN {X 0,Y 266.909,Z 786.593,A -85,B 0,C 180,E1 -19849.203,E2 -19849.203} C_VEL
LIN {X 0,Y 266.631,Z 804.51,A -85,B 0,C 180,E1 -19850.967,E2 -19850.967} C_VEL
LIN {X 0,Y 266.064,Z 824.543,A -85,B 0,C 180,E1 -19852.627,E2 -19852.627} C_VEL
LIN {X 0,Y 264.736,Z 845.359,A -85,B 0,C 180,E1 -19853.953,E2 -19853.953} C_VEL
LIN {X 0,Y 261.998,Z 864.865,A -85,B 0,C 180,E1 -19854.845,E2 -19854.845} C_VEL
LIN {X 0,Y 258.979,Z 878.824,A -85,B 0,C 180,E1 -19855.727,E2 -19855.727} C_VEL
LIN {X 0,Y 256.339,Z 888.672,A -85,B 0,C 180,E1 -19856.509,E2 -19856.509} C_VEL
LIN {X 0,Y 253.348,Z 898.495,A -85,B 0,C 180,E1 -19857.486,E2 -19857.486} C_VEL
LIN {X 0,Y 250.143,Z 908.222,A -85,B 0,C 180,E1 -19858.68,E2 -19858.68} C_VEL
LIN {X 0,Y 246.593,Z 917.69,A -85,B 0,C 180,E1 -19860.08,E2 -19860.08} C_VEL
LIN {X 0,Y 243.349,Z 925.825,A -85,B 0,C 180,E1 -19861.539,E2 -19861.539} C_VEL
LIN {X 0,Y 239.77,Z 934.521,A -85,B 0,C 180,E1 -19863.446,E2 -19863.446} C_VEL
LIN {X 0,Y 236.553,Z 941.963,A -85,B 0,C 180,E1 -19865.419,E2 -19865.419} C_VEL
LIN {X 0,Y 233.32,Z 949.447,A -85,B 0,C 180,E1 -19867.879,E2 -19867.879} C_VEL
LIN {X 0,Y 231.555,Z 953.842,A -85,B 0,C 180,E1 -19869.569,E2 -19869.569} C_VEL
LIN {X 0,Y 229.324,Z 959.3,A -85,B 0,C 180,E1 -19872.151,E2 -19872.151} C_VEL
LIN {X 0,Y 227.946,Z 963.72,A -85,B 0,C 180,E1 -19874.804,E2 -19874.804} C_VEL
LIN {X 0,Y 227.016,Z 967.149,A -85,B 0,C 180,E1 -19877.482,E2 -19877.482} C_VEL
LIN {X 0,Y 226.942,Z 971.961,A -85,B 0,C 180,E1 -19882.882,E2 -19882.882} C_VEL
LIN {X 0,Y 227.148,Z 973.813,A -85,B 0,C 180,E1 -19884.671,E2 -19884.671} C_VEL
LIN {X 0,Y 227.376,Z 975.185,A -85,B 0,C 180,E1 -19886.453,E2 -19886.453} C_VEL
LIN {X 0,Y 227.607,Z 976.125,A -85,B 0,C 180,E1 -19888.228,E2 -19888.228} C_VEL
LIN {X 0,Y 227.821,Z 976.637,A -85,B 0,C 180,E1 -19889.997,E2 -19889.997} C_VEL
LIN {X 0,Y 227.556,Z 976.618,A -85,B 0,C 180,E1 -19891.767,E2 -19891.767} C_VEL
LIN {X 0,Y 227.318,Z 976.168,A -85,B 0,C 180,E1 -19893.542,E2 -19893.542} C_VEL
LIN {X 0,Y 227.035,Z 975.301,A -85,B 0,C 180,E1 -19895.326,E2 -19895.326} C_VEL
LIN {X 0,Y 226.744,Z 973.855,A -85,B 0,C 180,E1 -19897.321,E2 -19897.321} C_VEL
LIN {X 0,Y 226.711,Z 970.144,A -85,B 0,C 180,E1 -19900.717,E2 -19900.717} C_VEL
LIN {X 0,Y 227.25,Z 966.092,A -85,B 0,C 180,E1 -19903.409,E2 -19903.409} C_VEL
LIN {X 0,Y 228.294,Z 960.941,A -85,B 0,C 180,E1 -19906.082,E2 -19906.082} C_VEL
LIN {X 0,Y 229.736,Z 955.158,A -85,B 0,C 180,E1 -19908.497,E2 -19908.497} C_VEL
LIN {X 0,Y 232.184,Z 946.743,A -85,B 0,C 180,E1 -19911.296,E2 -19911.296} C_VEL
LIN {X 0,Y 234.564,Z 938.876,A -85,B 0,C 180,E1 -19913.388,E2 -19913.388} C_VEL
LIN {X 0,Y 237.308,Z 929.413,A -85,B 0,C 180,E1 -19915.428,E2 -19915.428} C_VEL
LIN {X 0,Y 240.148,Z 918.972,A -85,B 0,C 180,E1 -19917.208,E2 -19917.208} C_VEL
LIN {X 0,Y 242.983,Z 907.487,A -85,B 0,C 180,E1 -19918.738,E2 -19918.738} C_VEL
LIN {X 0,Y 245.464,Z 895.635,A -85,B 0,C 180,E1 -19919.948,E2 -19919.948} C_VEL
LIN {X 0,Y 247.437,Z 882.738,A -85,B 0,C 180,E1 -19920.922,E2 -19920.922} C_VEL
LIN {X 0,Y 248.896,Z 869.237,A -85,B 0,C 180,E1 -19921.608,E2 -19921.608} C_VEL
LIN {X 0,Y 250.33,Z 838.74,A -85,B 0,C 180,E1 -19922.547,E2 -19922.547} C_VEL
LIN {X 0,Y 248.641,Z 812.62,A -85,B 0,C 180,E1 -19923.806,E2 -19923.806} C_VEL
LIN {X 0,Y 246.617,Z 790.828,A -85,B 0,C 180,E1 -19925.01,E2 -19925.01} C_VEL
LIN {X 0,Y 243.808,Z 771.175,A -85,B 0,C 180,E1 -19926.33,E2 -19926.33} C_VEL
LIN {X 0,Y 238.646,Z 759.471,A -85,B 0,C 180,E1 -19927.882,E2 -19927.882} C_VEL
LIN {X 0,Y 236.488,Z 754.493,A -85,B 0,C 180,E1 -19928.683,E2 -19928.683} C_VEL
LIN {X 0,Y 234.345,Z 745.816,A -85,B 0,C 180,E1 -19932.076,E2 -19932.076} C_VEL
LIN {X 0,Y 232.02,Z 737.271,A -85,B 0,C 180,E1 -19935.839,E2 -19935.839} C_VEL
LIN {X 0,Y 230.051,Z 730.945,A -85,B 0,C 180,E1 -19938.942,E2 -19938.942} C_VEL
LIN {X 0,Y 227.881,Z 724.158,A -85,B 0,C 180,E1 -19942.781,E2 -19942.781} C_VEL
LIN {X 0,Y 227.881,Z 724.088,A -85,B 0,C 180,E1 -19946.372,E2 -19946.372} C_VEL
LIN {X 0,Y 227.909,Z 724.098,A -85,B 0,C 180,E1 -19950.437,E2 -19950.437} C_VEL
LIN {X 0,Y 227.918,Z 724.089,A -85,B 0,C 180,E1 -19954.425,E2 -19954.425} C_VEL
LIN {X 0,Y 227.952,Z 724.081,A -85,B 0,C 180,E1 -19958.286,E2 -19958.286} C_VEL
LIN {X 0,Y 228.024,Z 724.07,A -85,B 0,C 180,E1 -19962.825,E2 -19962.825} C_VEL
LIN {X 0,Y 228.061,Z 724.067,A -85,B 0,C 180,E1 -19967.543,E2 -19967.543} C_VEL
LIN {X 0,Y 228.256,Z 724.038,A -85,B 0,C 180,E1 -19971.144,E2 -19971.144} C_VEL
LIN {X 0,Y 228.328,Z 724.042,A -85,B 0,C 180,E1 -19972.928,E2 -19972.928} C_VEL
LIN {X 0,Y 228.544,Z 724.017,A -85,B 0,C 180,E1 -19978.238,E2 -19978.238} C_VEL
LIN {X 0,Y 228.544,Z 724.013,A -85,B 0,C 180,E1 -19981.762,E2 -19981.762} C_VEL
LIN {X 0,Y 228.344,Z 724.04,A -85,B 0,C 180,E1 -19987.072,E2 -19987.072} C_VEL
LIN {X 0,Y 228.148,Z 724.068,A -85,B 0,C 180,E1 -19990.651,E2 -19990.651} C_VEL
LIN {X 0,Y 228.054,Z 724.079,A -85,B 0,C 180,E1 -19994.273,E2 -19994.273} C_VEL
LIN {X 0,Y 227.992,Z 724.086,A -85,B 0,C 180,E1 -19997.955,E2 -19997.955} C_VEL
LIN {X 0,Y 227.907,Z 724.075,A -85,B 0,C 180,E1 -20002.322,E2 -20002.322} C_VEL
LIN {X 0,Y 227.958,Z 724.325,A -85,B 0,C 180,E1 -20004.778,E2 -20004.778} C_VEL
LIN {X 0,Y 228.239,Z 725.478,A -85,B 0,C 180,E1 -20005.171,E2 -20005.171} C_VEL
LIN {X 0,Y 229.782,Z 728.084,A -85,B 0,C 180,E1 -20005.726,E2 -20005.726} C_VEL
LIN {X 0,Y 231.06,Z 729.322,A -85,B 0,C 180,E1 -20006.119,E2 -20006.119} C_VEL
LIN {X 0,Y 233.019,Z 732.555,A -85,B 0,C 180,E1 -20006.763,E2 -20006.763} C_VEL
LIN {X 0,Y 234.473,Z 734.486,A -85,B 0,C 180,E1 -20007.2,E2 -20007.2} C_VEL
LIN {X 0,Y 241.678,Z 745.712,A -85,B 0,C 180,E1 -20009.32,E2 -20009.32} C_VEL
LIN {X 0,Y 248.301,Z 757.225,A -85,B 0,C 180,E1 -20011.12,E2 -20011.12} C_VEL
LIN {X 0,Y 253.318,Z 767.358,A -85,B 0,C 180,E1 -20012.444,E2 -20012.444} C_VEL
LIN {X 0,Y 252.073,Z 803.703,A -85,B 0,C 180,E1 -20013.584,E2 -20013.584} C_VEL
LIN {X 0,Y 251.655,Z 817.331,A -85,B 0,C 180,E1 -20014.182,E2 -20014.182} C_VEL
LIN {X 0,Y 250.745,Z 829.95,A -85,B 0,C 180,E1 -20015.054,E2 -20015.054} C_VEL
LIN {X 0,Y 249.299,Z 841.989,A -85,B 0,C 180,E1 -20016.184,E2 -20016.184} C_VEL
LIN {X 0,Y 247.367,Z 853.684,A -85,B 0,C 180,E1 -20017.631,E2 -20017.631} C_VEL
LIN {X 0,Y 245.176,Z 864.184,A -85,B 0,C 180,E1 -20019.294,E2 -20019.294} C_VEL
LIN {X 0,Y 242.829,Z 873.78,A -85,B 0,C 180,E1 -20021.197,E2 -20021.197} C_VEL
LIN {X 0,Y 240.612,Z 881.57,A -85,B 0,C 180,E1 -20023.099,E2 -20023.099} C_VEL
LIN {X 0,Y 238.106,Z 889.49,A -85,B 0,C 180,E1 -20025.496,E2 -20025.496} C_VEL
LIN {X 0,Y 235.746,Z 896.393,A -85,B 0,C 180,E1 -20028.185,E2 -20028.185} C_VEL
LIN {X 0,Y 233.712,Z 901.708,A -85,B 0,C 180,E1 -20030.843,E2 -20030.843} C_VEL
LIN {X 0,Y 231.831,Z 906.097,A -85,B 0,C 180,E1 -20033.765,E2 -20033.765} C_VEL
LIN {X 0,Y 230.513,Z 909.117,A -85,B 0,C 180,E1 -20036.719,E2 -20036.719} C_VEL
LIN {X 0,Y 229.73,Z 910.577,A -85,B 0,C 180,E1 -20038.937,E2 -20038.937} C_VEL
LIN {X 0,Y 229.284,Z 911.285,A -85,B 0,C 180,E1 -20040.634,E2 -20040.634} C_VEL
LIN {X 0,Y 228.894,Z 911.613,A -85,B 0,C 180,E1 -20042.928,E2 -20042.928} C_VEL
LIN {X 0,Y 228.662,Z 910.893,A -85,B 0,C 180,E1 -20046.452,E2 -20046.452} C_VEL
LIN {X 0,Y 228.759,Z 909.806,A -85,B 0,C 180,E1 -20048.37,E2 -20048.37} C_VEL
LIN {X 0,Y 229.376,Z 906.732,A -85,B 0,C 180,E1 -20051.776,E2 -20051.776} C_VEL
LIN {X 0,Y 230.452,Z 902.283,A -85,B 0,C 180,E1 -20054.979,E2 -20054.979} C_VEL
LIN {X 0,Y 231.872,Z 896.148,A -85,B 0,C 180,E1 -20058.197,E2 -20058.197} C_VEL
LIN {X 0,Y 233.454,Z 889.361,A -85,B 0,C 180,E1 -20060.909,E2 -20060.909} C_VEL
LIN {X 0,Y 235.328,Z 880.888,A -85,B 0,C 180,E1 -20063.572,E2 -20063.572} C_VEL
LIN {X 0,Y 237.157,Z 872.221,A -85,B 0,C 180,E1 -20065.754,E2 -20065.754} C_VEL
LIN {X 0,Y 238.918,Z 862.77,A -85,B 0,C 180,E1 -20067.683,E2 -20067.683} C_VEL
LIN {X 0,Y 240.604,Z 852.441,A -85,B 0,C 180,E1 -20069.375,E2 -20069.375} C_VEL
LIN {X 0,Y 242.113,Z 841.264,A -85,B 0,C 180,E1 -20070.834,E2 -20070.834} C_VEL
LIN {X 0,Y 243.391,Z 828.984,A -85,B 0,C 180,E1 -20072.071,E2 -20072.071} C_VEL
LIN {X 0,Y 244.193,Z 815.566,A -85,B 0,C 180,E1 -20073.044,E2 -20073.044} C_VEL
LIN {X 0,Y 244.582,Z 802.475,A -85,B 0,C 180,E1 -20073.657,E2 -20073.657} C_VEL
LIN {X 0,Y 245.519,Z 760.044,A -85,B 0,C 180,E1 -20074.985,E2 -20074.985} C_VEL
LIN {X 0,Y 239.215,Z 746.095,A -85,B 0,C 180,E1 -20076.253,E2 -20076.253} C_VEL
LIN {X 0,Y 229.449,Z 727.137,A -85,B 0,C 180,E1 -20078.281,E2 -20078.281} C_VEL
LIN {X 0,Y 228.412,Z 724.8,A -85,B 0,C 180,E1 -20078.574,E2 -20078.574} C_VEL
LIN {X 0,Y 228.266,Z 724.097,A -85,B 0,C 180,E1 -20078.99,E2 -20078.99} C_VEL
LIN {X 0,Y 228.011,Z 724.069,A -85,B 0,C 180,E1 -20084.278,E2 -20084.278} C_VEL
LIN {X 0,Y 227.932,Z 724.089,A -85,B 0,C 180,E1 -20087.962,E2 -20087.962} C_VEL
LIN {X 0,Y 227.898,Z 724.095,A -85,B 0,C 180,E1 -20092.307,E2 -20092.307} C_VEL
LIN {X 0,Y 227.876,Z 724.07,A -85,B 0,C 180,E1 -20096.567,E2 -20096.567} C_VEL
LIN {X 0,Y 227.876,Z 724.1,A -85,B 0,C 180,E1 -20100.281,E2 -20100.281} C_VEL
LIN {X 0,Y 227.879,Z 724.064,A -85,B 0,C 180,E1 -20103.723,E2 -20103.723} C_VEL
LIN {X 0,Y 227.847,Z 724.094,A -85,B 0,C 180,E1 -20108.093,E2 -20108.093} C_VEL
LIN {X 0,Y 227.792,Z 724.11,A -85,B 0,C 180,E1 -20112.75,E2 -20112.75} C_VEL
LIN {X 0,Y 227.793,Z 724.109,A -85,B 0,C 180,E1 -20117.253,E2 -20117.253} C_VEL
LIN {X 0,Y 227.86,Z 724.335,A -85,B 0,C 180,E1 -20119.057,E2 -20119.057} C_VEL
LIN {X 0,Y 228.11,Z 725.317,A -85,B 0,C 180,E1 -20119.314,E2 -20119.314} C_VEL
LIN {X 0,Y 237.609,Z 752.568,A -85,B 0,C 180,E1 -20121.229,E2 -20121.229} C_VEL
LIN {X 0,Y 235.922,Z 804.009,A -85,B 0,C 180,E1 -20123.473,E2 -20123.473} C_VEL
LIN {X 0,Y 235.522,Z 814.72,A -85,B 0,C 180,E1 -20124.153,E2 -20124.153} C_VEL
LIN {X 0,Y 234.805,Z 825.765,A -85,B 0,C 180,E1 -20125.079,E2 -20125.079} C_VEL
LIN {X 0,Y 233.969,Z 836.616,A -85,B 0,C 180,E1 -20126.24,E2 -20126.24} C_VEL
LIN {X 0,Y 233.188,Z 845.942,A -85,B 0,C 180,E1 -20127.462,E2 -20127.462} C_VEL
LIN {X 0,Y 232.335,Z 854.678,A -85,B 0,C 180,E1 -20128.822,E2 -20128.822} C_VEL
LIN {X 0,Y 231.477,Z 863.424,A -85,B 0,C 180,E1 -20130.437,E2 -20130.437} C_VEL
LIN {X 0,Y 230.596,Z 871.754,A -85,B 0,C 180,E1 -20132.255,E2 -20132.255} C_VEL
LIN {X 0,Y 229.762,Z 879.169,A -85,B 0,C 180,E1 -20134.158,E2 -20134.158} C_VEL
LIN {X 0,Y 229.229,Z 885.407,A -85,B 0,C 180,E1 -20136.031,E2 -20136.031} C_VEL
LIN {X 0,Y 228.66,Z 891.873,A -85,B 0,C 180,E1 -20138.356,E2 -20138.356} C_VEL
LIN {X 0,Y 228.356,Z 896.299,A -85,B 0,C 180,E1 -20140.211,E2 -20140.211} C_VEL
LIN {X 0,Y 228.145,Z 901.24,A -85,B 0,C 180,E1 -20142.745,E2 -20142.745} C_VEL
LIN {X 0,Y 228.239,Z 905.686,A -85,B 0,C 180,E1 -20145.739,E2 -20145.739} C_VEL
LIN {X 0,Y 228.499,Z 907.836,A -85,B 0,C 180,E1 -20147.566,E2 -20147.566} C_VEL
LIN {X 0,Y 229.413,Z 910.62,A -85,B 0,C 180,E1 -20151.189,E2 -20151.189} C_VEL
LIN {X 0,Y 230.144,Z 911.36,A -85,B 0,C 180,E1 -20152.984,E2 -20152.984} C_VEL
LIN {X 0,Y 231.009,Z 911.63,A -85,B 0,C 180,E1 -20154.763,E2 -20154.763} C_VEL
LIN {X 0,Y 233.181,Z 910.901,A -85,B 0,C 180,E1 -20158.273,E2 -20158.273} C_VEL
LIN {X 0,Y 235.958,Z 908.347,A -85,B 0,C 180,E1 -20161.707,E2 -20161.707} C_VEL
LIN {X 0,Y 238.414,Z 905.327,A -85,B 0,C 180,E1 -20164.226,E2 -20164.226} C_VEL
LIN {X 0,Y 240.157,Z 903.017,A -85,B 0,C 180,E1 -20165.722,E2 -20165.722} C_VEL
LIN {X 0,Y 243.975,Z 896.74,A -85,B 0,C 180,E1 -20168.698,E2 -20168.698} C_VEL
LIN {X 0,Y 246.811,Z 891.476,A -85,B 0,C 180,E1 -20170.666,E2 -20170.666} C_VEL
LIN {X 0,Y 249.919,Z 885.078,A -85,B 0,C 180,E1 -20172.588,E2 -20172.588} C_VEL
LIN {X 0,Y 253.155,Z 877.438,A -85,B 0,C 180,E1 -20174.448,E2 -20174.448} C_VEL
LIN {X 0,Y 254.333,Z 873.53,A -85,B 0,C 180,E1 -20175.414,E2 -20175.414} C_VEL
LIN {X 0,Y 254.873,Z 867.381,A -85,B 0,C 180,E1 -20177.181,E2 -20177.181} C_VEL
LIN {X 0,Y 255.465,Z 860.803,A -85,B 0,C 180,E1 -20178.822,E2 -20178.822} C_VEL
LIN {X 0,Y 256.48,Z 856.147,A -85,B 0,C 180,E1 -20179.583,E2 -20179.583} C_VEL
LIN {X 0,Y 259.234,Z 845.594,A -85,B 0,C 180,E1 -20180.844,E2 -20180.844} C_VEL
LIN {X 0,Y 261.44,Z 834.776,A -85,B 0,C 180,E1 -20181.9,E2 -20181.9} C_VEL
LIN {X 0,Y 263.152,Z 824.131,A -85,B 0,C 180,E1 -20182.714,E2 -20182.714} C_VEL
LIN {X 0,Y 265.653,Z 803.155,A -85,B 0,C 180,E1 -20183.882,E2 -20183.882} C_VEL
LIN {X 0,Y 268.026,Z 785.149,A -85,B 0,C 180,E1 -20184.735,E2 -20184.735} C_VEL
LIN {X 0,Y 265.729,Z 780.47,A -85,B 0,C 180,E1 -20186.411,E2 -20186.411} C_VEL
LIN {X 0,Y 263.166,Z 775.316,A -85,B 0,C 180,E1 -20188.731,E2 -20188.731} C_VEL
LIN {X 0,Y 261.136,Z 771.591,A -85,B 0,C 180,E1 -20191.157,E2 -20191.157} C_VEL
LIN {X 0,Y 259.414,Z 768.832,A -85,B 0,C 180,E1 -20194.509,E2 -20194.509} C_VEL
LIN {X 0,Y 259.149,Z 768.515,A -85,B 0,C 180,E1 -20195.549,E2 -20195.549} C_VEL
LIN {X 0,Y 258.878,Z 769.252,A -85,B 0,C 180,E1 -20198.311,E2 -20198.311} C_VEL
LIN {X 0,Y 259.783,Z 771.357,A -85,B 0,C 180,E1 -20201.402,E2 -20201.402} C_VEL
LIN {X 0,Y 261.666,Z 775.545,A -85,B 0,C 180,E1 -20204.434,E2 -20204.434} C_VEL
LIN {X 0,Y 262.004,Z 777.123,A -85,B 0,C 180,E1 -20204.979,E2 -20204.979} C_VEL
LIN {X 0,Y 263.092,Z 785.776,A -85,B 0,C 180,E1 -20207.063,E2 -20207.063} C_VEL
LIN {X 0,Y 263.75,Z 790.5,A -85,B 0,C 180,E1 -20208.09,E2 -20208.09} C_VEL
LIN {X 0,Y 263.155,Z 807.988,A -85,B 0,C 180,E1 -20209.828,E2 -20209.828} C_VEL
LIN {X 0,Y 262.316,Z 826.763,A -85,B 0,C 180,E1 -20211.404,E2 -20211.404} C_VEL
LIN {X 0,Y 260.771,Z 846.664,A -85,B 0,C 180,E1 -20212.701,E2 -20212.701} C_VEL
LIN {X 0,Y 257.972,Z 864.472,A -85,B 0,C 180,E1 -20213.539,E2 -20213.539} C_VEL
LIN {X 0,Y 255.218,Z 876.518,A -85,B 0,C 180,E1 -20214.304,E2 -20214.304} C_VEL
LIN {X 0,Y 252.147,Z 887.26,A -85,B 0,C 180,E1 -20215.15,E2 -20215.15} C_VEL
LIN {X 0,Y 248.515,Z 898.524,A -85,B 0,C 180,E1 -20216.287,E2 -20216.287} C_VEL
LIN {X 0,Y 245.112,Z 907.951,A -85,B 0,C 180,E1 -20217.476,E2 -20217.476} C_VEL
LIN {X 0,Y 241.425,Z 917.144,A -85,B 0,C 180,E1 -20218.886,E2 -20218.886} C_VEL
LIN {X 0,Y 238.029,Z 925.135,A -85,B 0,C 180,E1 -20220.357,E2 -20220.357} C_VEL
LIN {X 0,Y 234.169,Z 933.688,A -85,B 0,C 180,E1 -20222.275,E2 -20222.275} C_VEL
LIN {X 0,Y 230.768,Z 940.981,A -85,B 0,C 180,E1 -20224.277,E2 -20224.277} C_VEL
LIN {X 0,Y 227.833,Z 947.301,A -85,B 0,C 180,E1 -20226.356,E2 -20226.356} C_VEL
LIN {X 0,Y 224.885,Z 953.638,A -85,B 0,C 180,E1 -20228.934,E2 -20228.934} C_VEL
LIN {X 0,Y 222.533,Z 958.858,A -85,B 0,C 180,E1 -20231.587,E2 -20231.587} C_VEL
LIN {X 0,Y 221.043,Z 963.085,A -85,B 0,C 180,E1 -20234.318,E2 -20234.318} C_VEL
LIN {X 0,Y 220.02,Z 966.359,A -85,B 0,C 180,E1 -20237.077,E2 -20237.077} C_VEL
LIN {X 0,Y 219.881,Z 970.803,A -85,B 0,C 180,E1 -20242.652,E2 -20242.652} C_VEL
LIN {X 0,Y 220.089,Z 972.699,A -85,B 0,C 180,E1 -20244.5,E2 -20244.5} C_VEL
LIN {X 0,Y 220.319,Z 974.096,A -85,B 0,C 180,E1 -20246.339,E2 -20246.339} C_VEL
LIN {X 0,Y 220.557,Z 975.058,A -85,B 0,C 180,E1 -20248.171,E2 -20248.171} C_VEL
LIN {X 0,Y 220.788,Z 975.592,A -85,B 0,C 180,E1 -20249.997,E2 -20249.997} C_VEL
LIN {X 0,Y 220.504,Z 975.61,A -85,B 0,C 180,E1 -20251.824,E2 -20251.824} C_VEL
LIN {X 0,Y 220.258,Z 975.178,A -85,B 0,C 180,E1 -20253.656,E2 -20253.656} C_VEL
LIN {X 0,Y 219.935,Z 974.322,A -85,B 0,C 180,E1 -20255.498,E2 -20255.498} C_VEL
LIN {X 0,Y 219.696,Z 973.026,A -85,B 0,C 180,E1 -20257.395,E2 -20257.395} C_VEL
LIN {X 0,Y 219.606,Z 970.357,A -85,B 0,C 180,E1 -20260.135,E2 -20260.135} C_VEL
LIN {X 0,Y 219.999,Z 966.678,A -85,B 0,C 180,E1 -20262.919,E2 -20262.919} C_VEL
LIN {X 0,Y 220.986,Z 961.961,A -85,B 0,C 180,E1 -20265.681,E2 -20265.681} C_VEL
LIN {X 0,Y 222.416,Z 956.075,A -85,B 0,C 180,E1 -20268.417,E2 -20268.417} C_VEL
LIN {X 0,Y 224.695,Z 948.876,A -85,B 0,C 180,E1 -20271.078,E2 -20271.078} C_VEL
LIN {X 0,Y 227.474,Z 939.982,A -85,B 0,C 180,E1 -20273.678,E2 -20273.678} C_VEL
LIN {X 0,Y 230.312,Z 930.958,A -85,B 0,C 180,E1 -20275.772,E2 -20275.772} C_VEL
LIN {X 0,Y 233.5,Z 919.94,A -85,B 0,C 180,E1 -20277.806,E2 -20277.806} C_VEL
LIN {X 0,Y 236.439,Z 908.964,A -85,B 0,C 180,E1 -20279.367,E2 -20279.367} C_VEL
LIN {X 0,Y 239.187,Z 896.754,A -85,B 0,C 180,E1 -20280.696,E2 -20280.696} C_VEL
LIN {X 0,Y 241.341,Z 883.758,A -85,B 0,C 180,E1 -20281.766,E2 -20281.766} C_VEL
LIN {X 0,Y 242.983,Z 870.328,A -85,B 0,C 180,E1 -20282.501,E2 -20282.501} C_VEL
LIN {X 0,Y 244.116,Z 850.714,A -85,B 0,C 180,E1 -20283.158,E2 -20283.158} C_VEL
LIN {X 0,Y 244.549,Z 838.509,A -85,B 0,C 180,E1 -20283.548,E2 -20283.548} C_VEL
LIN {X 0,Y 243.061,Z 814.168,A -85,B 0,C 180,E1 -20284.764,E2 -20284.764} C_VEL
LIN {X 0,Y 241.164,Z 792.59,A -85,B 0,C 180,E1 -20285.991,E2 -20285.991} C_VEL
LIN {X 0,Y 238.635,Z 774.189,A -85,B 0,C 180,E1 -20287.264,E2 -20287.264} C_VEL
LIN {X 0,Y 233.884,Z 763.32,A -85,B 0,C 180,E1 -20288.79,E2 -20288.79} C_VEL
LIN {X 0,Y 231.031,Z 757.39,A -85,B 0,C 180,E1 -20289.739,E2 -20289.739} C_VEL
LIN {X 0,Y 228.983,Z 752.955,A -85,B 0,C 180,E1 -20290.52,E2 -20290.52} C_VEL
LIN {X 0,Y 226.931,Z 744.92,A -85,B 0,C 180,E1 -20293.919,E2 -20293.919} C_VEL
LIN {X 0,Y 224.659,Z 736.927,A -85,B 0,C 180,E1 -20297.733,E2 -20297.733} C_VEL
LIN {X 0,Y 222.154,Z 729.307,A -85,B 0,C 180,E1 -20301.911,E2 -20301.911} C_VEL
LIN {X 0,Y 220.841,Z 725.024,A -85,B 0,C 180,E1 -20304.634,E2 -20304.634} C_VEL
LIN {X 0,Y 220.858,Z 724.97,A -85,B 0,C 180,E1 -20309.394,E2 -20309.394} C_VEL
LIN {X 0,Y 220.885,Z 724.972,A -85,B 0,C 180,E1 -20313.548,E2 -20313.548} C_VEL
LIN {X 0,Y 220.868,Z 724.969,A -85,B 0,C 180,E1 -20317.553,E2 -20317.553} C_VEL
LIN {X 0,Y 220.974,Z 724.948,A -85,B 0,C 180,E1 -20322.57,E2 -20322.57} C_VEL
LIN {X 0,Y 221,Z 724.945,A -85,B 0,C 180,E1 -20327.138,E2 -20327.138} C_VEL
LIN {X 0,Y 221.193,Z 724.918,A -85,B 0,C 180,E1 -20330.859,E2 -20330.859} C_VEL
LIN {X 0,Y 221.261,Z 724.919,A -85,B 0,C 180,E1 -20332.701,E2 -20332.701} C_VEL
LIN {X 0,Y 221.502,Z 724.894,A -85,B 0,C 180,E1 -20338.182,E2 -20338.182} C_VEL
LIN {X 0,Y 221.502,Z 724.89,A -85,B 0,C 180,E1 -20341.819,E2 -20341.819} C_VEL
LIN {X 0,Y 221.279,Z 724.918,A -85,B 0,C 180,E1 -20347.299,E2 -20347.299} C_VEL
LIN {X 0,Y 221.096,Z 724.943,A -85,B 0,C 180,E1 -20350.995,E2 -20350.995} C_VEL
LIN {X 0,Y 221.006,Z 724.948,A -85,B 0,C 180,E1 -20356.631,E2 -20356.631} C_VEL
LIN {X 0,Y 220.874,Z 724.971,A -85,B 0,C 180,E1 -20360.488,E2 -20360.488} C_VEL
LIN {X 0,Y 220.897,Z 725.245,A -85,B 0,C 180,E1 -20362.819,E2 -20362.819} C_VEL
LIN {X 0,Y 221.174,Z 726.354,A -85,B 0,C 180,E1 -20363.204,E2 -20363.204} C_VEL
LIN {X 0,Y 222.68,Z 728.89,A -85,B 0,C 180,E1 -20363.797,E2 -20363.797} C_VEL
LIN {X 0,Y 224.293,Z 730.489,A -85,B 0,C 180,E1 -20364.346,E2 -20364.346} C_VEL
LIN {X 0,Y 226.354,Z 733.751,A -85,B 0,C 180,E1 -20365.088,E2 -20365.088} C_VEL
LIN {X 0,Y 227.708,Z 735.528,A -85,B 0,C 180,E1 -20365.54,E2 -20365.54} C_VEL
LIN {X 0,Y 233.31,Z 743.923,A -85,B 0,C 180,E1 -20367.347,E2 -20367.347} C_VEL
LIN {X 0,Y 239.759,Z 754.515,A -85,B 0,C 180,E1 -20369.278,E2 -20369.278} C_VEL
LIN {X 0,Y 246.096,Z 766.309,A -85,B 0,C 180,E1 -20371.053,E2 -20371.053} C_VEL
LIN {X 0,Y 247.689,Z 769.865,A -85,B 0,C 180,E1 -20371.5,E2 -20371.5} C_VEL
LIN {X 0,Y 246.412,Z 805.249,A -85,B 0,C 180,E1 -20372.643,E2 -20372.643} C_VEL
LIN {X 0,Y 245.955,Z 818.505,A -85,B 0,C 180,E1 -20373.247,E2 -20373.247} C_VEL
LIN {X 0,Y 244.955,Z 831.38,A -85,B 0,C 180,E1 -20374.165,E2 -20374.165} C_VEL
LIN {X 0,Y 243.494,Z 842.779,A -85,B 0,C 180,E1 -20375.259,E2 -20375.259} C_VEL
LIN {X 0,Y 241.683,Z 853.318,A -85,B 0,C 180,E1 -20376.557,E2 -20376.557} C_VEL
LIN {X 0,Y 239.418,Z 864.128,A -85,B 0,C 180,E1 -20378.262,E2 -20378.262} C_VEL
LIN {X 0,Y 237.045,Z 873.369,A -85,B 0,C 180,E1 -20380.076,E2 -20380.076} C_VEL
LIN {X 0,Y 234.555,Z 881.854,A -85,B 0,C 180,E1 -20382.137,E2 -20382.137} C_VEL
LIN {X 0,Y 231.821,Z 890.225,A -85,B 0,C 180,E1 -20384.691,E2 -20384.691} C_VEL
LIN {X 0,Y 229.165,Z 897.481,A -85,B 0,C 180,E1 -20387.574,E2 -20387.574} C_VEL
LIN {X 0,Y 227.035,Z 902.774,A -85,B 0,C 180,E1 -20390.306,E2 -20390.306} C_VEL
LIN {X 0,Y 224.886,Z 907.466,A -85,B 0,C 180,E1 -20393.578,E2 -20393.578} C_VEL
LIN {X 0,Y 223.95,Z 909.515,A -85,B 0,C 180,E1 -20395.61,E2 -20395.61} C_VEL
LIN {X 0,Y 222.885,Z 911.462,A -85,B 0,C 180,E1 -20398.361,E2 -20398.361} C_VEL
LIN {X 0,Y 222.044,Z 912.573,A -85,B 0,C 180,E1 -20401.659,E2 -20401.659} C_VEL
LIN {X 0,Y 221.769,Z 912.609,A -85,B 0,C 180,E1 -20403.665,E2 -20403.665} C_VEL
LIN {X 0,Y 221.653,Z 911.673,A -85,B 0,C 180,E1 -20406.856,E2 -20406.856} C_VEL
LIN {X 0,Y 221.903,Z 909.895,A -85,B 0,C 180,E1 -20409.614,E2 -20409.614} C_VEL
LIN {X 0,Y 222.565,Z 906.938,A -85,B 0,C 180,E1 -20412.546,E2 -20412.546} C_VEL
LIN {X 0,Y 223.574,Z 902.854,A -85,B 0,C 180,E1 -20415.438,E2 -20415.438} C_VEL
LIN {X 0,Y 224.829,Z 897.577,A -85,B 0,C 180,E1 -20418.28,E2 -20418.28} C_VEL
LIN {X 0,Y 226.465,Z 890.918,A -85,B 0,C 180,E1 -20421.076,E2 -20421.076} C_VEL
LIN {X 0,Y 228.414,Z 882.55,A -85,B 0,C 180,E1 -20423.82,E2 -20423.82} C_VEL
LIN {X 0,Y 230.24,Z 874.035,A -85,B 0,C 180,E1 -20426.064,E2 -20426.064} C_VEL
LIN {X 0,Y 232.066,Z 864.926,A -85,B 0,C 180,E1 -20428.013,E2 -20428.013} C_VEL
LIN {X 0,Y 233.856,Z 854.681,A -85,B 0,C 180,E1 -20429.787,E2 -20429.787} C_VEL
LIN {X 0,Y 235.4,Z 843.811,A -85,B 0,C 180,E1 -20431.286,E2 -20431.286} C_VEL
LIN {X 0,Y 236.848,Z 830.826,A -85,B 0,C 180,E1 -20432.66,E2 -20432.66} C_VEL
LIN {X 0,Y 237.735,Z 817.841,A -85,B 0,C 180,E1 -20433.658,E2 -20433.658} C_VEL
LIN {X 0,Y 238.179,Z 803.942,A -85,B 0,C 180,E1 -20434.349,E2 -20434.349} C_VEL
LIN {X 0,Y 239.203,Z 762.024,A -85,B 0,C 180,E1 -20435.694,E2 -20435.694} C_VEL
LIN {X 0,Y 233.604,Z 749.644,A -85,B 0,C 180,E1 -20436.871,E2 -20436.871} C_VEL
LIN {X 0,Y 224.36,Z 731.532,A -85,B 0,C 180,E1 -20438.86,E2 -20438.86} C_VEL
LIN {X 0,Y 221.448,Z 726.055,A -85,B 0,C 180,E1 -20439.541,E2 -20439.541} C_VEL
LIN {X 0,Y 221.231,Z 725.197,A -85,B 0,C 180,E1 -20439.807,E2 -20439.807} C_VEL
LIN {X 0,Y 221.065,Z 724.937,A -85,B 0,C 180,E1 -20440.999,E2 -20440.999} C_VEL
LIN {X 0,Y 220.981,Z 724.955,A -85,B 0,C 180,E1 -20446.635,E2 -20446.635} C_VEL
LIN {X 0,Y 220.853,Z 724.953,A -85,B 0,C 180,E1 -20450.493,E2 -20450.493} C_VEL
LIN {X 0,Y 220.809,Z 724.969,A -85,B 0,C 180,E1 -20454.445,E2 -20454.445} C_VEL
LIN {X 0,Y 220.798,Z 724.967,A -85,B 0,C 180,E1 -20458.522,E2 -20458.522} C_VEL
LIN {X 0,Y 220.817,Z 724.956,A -85,B 0,C 180,E1 -20462.759,E2 -20462.759} C_VEL
LIN {X 0,Y 220.809,Z 724.961,A -85,B 0,C 180,E1 -20467.277,E2 -20467.277} C_VEL
LIN {X 0,Y 220.755,Z 724.988,A -85,B 0,C 180,E1 -20471.959,E2 -20471.959} C_VEL
LIN {X 0,Y 220.76,Z 724.987,A -85,B 0,C 180,E1 -20475.542,E2 -20475.542} C_VEL
LIN {X 0,Y 220.817,Z 725.137,A -85,B 0,C 180,E1 -20478.524,E2 -20478.524} C_VEL
LIN {X 0,Y 221.037,Z 726.123,A -85,B 0,C 180,E1 -20478.828,E2 -20478.828} C_VEL
LIN {X 0,Y 230.748,Z 754.04,A -85,B 0,C 180,E1 -20480.873,E2 -20480.873} C_VEL
LIN {X 0,Y 228.93,Z 805.248,A -85,B 0,C 180,E1 -20483.184,E2 -20483.184} C_VEL
LIN {X 0,Y 228.493,Z 816.045,A -85,B 0,C 180,E1 -20483.896,E2 -20483.896} C_VEL
LIN {X 0,Y 227.813,Z 826.46,A -85,B 0,C 180,E1 -20484.794,E2 -20484.794} C_VEL
LIN {X 0,Y 227.037,Z 836.418,A -85,B 0,C 180,E1 -20485.87,E2 -20485.87} C_VEL
LIN {X 0,Y 226.218,Z 846.058,A -85,B 0,C 180,E1 -20487.142,E2 -20487.142} C_VEL
LIN {X 0,Y 225.247,Z 856.111,A -85,B 0,C 180,E1 -20488.753,E2 -20488.753} C_VEL
LIN {X 0,Y 224.343,Z 864.904,A -85,B 0,C 180,E1 -20490.446,E2 -20490.446} C_VEL
LIN {X 0,Y 223.421,Z 873.286,A -85,B 0,C 180,E1 -20492.355,E2 -20492.355} C_VEL
LIN {X 0,Y 222.612,Z 880.45,A -85,B 0,C 180,E1 -20494.272,E2 -20494.272} C_VEL
LIN {X 0,Y 222.047,Z 886.922,A -85,B 0,C 180,E1 -20496.303,E2 -20496.303} C_VEL
LIN {X 0,Y 221.528,Z 893.102,A -85,B 0,C 180,E1 -20498.602,E2 -20498.602} C_VEL
LIN {X 0,Y 221.254,Z 897.538,A -85,B 0,C 180,E1 -20500.517,E2 -20500.517} C_VEL
LIN {X 0,Y 221.047,Z 902.847,A -85,B 0,C 180,E1 -20503.372,E2 -20503.372} C_VEL
LIN {X 0,Y 221.241,Z 906.924,A -85,B 0,C 180,E1 -20506.217,E2 -20506.217} C_VEL
LIN {X 0,Y 221.806,Z 910,A -85,B 0,C 180,E1 -20509.2,E2 -20509.2} C_VEL
LIN {X 0,Y 222.284,Z 911.345,A -85,B 0,C 180,E1 -20510.904,E2 -20510.904} C_VEL
LIN {X 0,Y 222.987,Z 912.283,A -85,B 0,C 180,E1 -20512.757,E2 -20512.757} C_VEL
LIN {X 0,Y 223.885,Z 912.784,A -85,B 0,C 180,E1 -20514.596,E2 -20514.596} C_VEL
LIN {X 0,Y 225.226,Z 912.785,A -85,B 0,C 180,E1 -20516.94,E2 -20516.94} C_VEL
LIN {X 0,Y 227.47,Z 911.663,A -85,B 0,C 180,E1 -20520,E2 -20520} C_VEL
LIN {X 0,Y 228.989,Z 910.52,A -85,B 0,C 180,E1 -20521.758,E2 -20521.758} C_VEL
LIN {X 0,Y 231.546,Z 907.859,A -85,B 0,C 180,E1 -20524.352,E2 -20524.352} C_VEL
LIN {X 0,Y 234.542,Z 904.1,A -85,B 0,C 180,E1 -20526.884,E2 -20526.884} C_VEL
LIN {X 0,Y 237.91,Z 899.172,A -85,B 0,C 180,E1 -20529.35,E2 -20529.35} C_VEL
LIN {X 0,Y 241.501,Z 892.931,A -85,B 0,C 180,E1 -20531.754,E2 -20531.754} C_VEL
LIN {X 0,Y 244.808,Z 886.561,A -85,B 0,C 180,E1 -20533.7,E2 -20533.7} C_VEL
LIN {X 0,Y 248.301,Z 878.967,A -85,B 0,C 180,E1 -20535.597,E2 -20535.597} C_VEL
LIN {X 0,Y 251.187,Z 871.787,A -85,B 0,C 180,E1 -20537.084,E2 -20537.084} C_VEL
LIN {X 0,Y 254.473,Z 862.464,A -85,B 0,C 180,E1 -20538.671,E2 -20538.671} C_VEL
LIN {X 0,Y 256.48,Z 856.147,A -85,B 0,C 180,E1 -20539.583,E2 -20539.583} C_VEL
LIN {X 0,Y 257.539,Z 851.317,A -85,B 0,C 180,E1 -20540.31,E2 -20540.31} C_VEL
LIN {X 0,Y 257.946,Z 843.811,A -85,B 0,C 180,E1 -20541.755,E2 -20541.755} C_VEL
LIN {X 0,Y 258.243,Z 836.024,A -85,B 0,C 180,E1 -20543.093,E2 -20543.093} C_VEL
LIN {X 0,Y 258.881,Z 830.775,A -85,B 0,C 180,E1 -20543.651,E2 -20543.651} C_VEL
LIN {X 0,Y 261.024,Z 815.393,A -85,B 0,C 180,E1 -20544.638,E2 -20544.638} C_VEL
LIN {X 0,Y 263.83,Z 794.427,A -85,B 0,C 180,E1 -20545.694,E2 -20545.694} C_VEL
LIN {X 0,Y 264.548,Z 789.218,A -85,B 0,C 180,E1 -20545.955,E2 -20545.955} C_VEL
LIN {X 0,Y 262.009,Z 783.856,A -85,B 0,C 180,E1 -20548.163,E2 -20548.163} C_VEL
LIN {X 0,Y 260.741,Z 781.321,A -85,B 0,C 180,E1 -20549.528,E2 -20549.528} C_VEL
LIN {X 0,Y 259.329,Z 778.336,A -85,B 0,C 180,E1 -20551.452,E2 -20551.452} C_VEL
LIN {X 0,Y 257.718,Z 775.506,A -85,B 0,C 180,E1 -20555.101,E2 -20555.101} C_VEL
LIN {X 0,Y 257.308,Z 776.013,A -85,B 0,C 180,E1 -20557.89,E2 -20557.89} C_VEL
LIN {X 0,Y 258.002,Z 777.998,A -85,B 0,C 180,E1 -20560.955,E2 -20560.955} C_VEL
LIN {X 0,Y 259.636,Z 781.985,A -85,B 0,C 180,E1 -20563.949,E2 -20563.949} C_VEL
LIN {X 0,Y 260.356,Z 789.978,A -85,B 0,C 180,E1 -20565.946,E2 -20565.946} C_VEL
LIN {X 0,Y 260.84,Z 794.8,A -85,B 0,C 180,E1 -20566.97,E2 -20566.97} C_VEL
LIN {X 0,Y 259.913,Z 811.059,A -85,B 0,C 180,E1 -20568.603,E2 -20568.603} C_VEL
LIN {X 0,Y 258.813,Z 828.537,A -85,B 0,C 180,E1 -20570.102,E2 -20570.102} C_VEL
LIN {X 0,Y 257.104,Z 847.784,A -85,B 0,C 180,E1 -20571.376,E2 -20571.376} C_VEL
LIN {X 0,Y 254.255,Z 863.934,A -85,B 0,C 180,E1 -20572.177,E2 -20572.177} C_VEL
LIN {X 0,Y 251.327,Z 875.627,A -85,B 0,C 180,E1 -20572.915,E2 -20572.915} C_VEL
LIN {X 0,Y 248.181,Z 886.244,A -85,B 0,C 180,E1 -20573.759,E2 -20573.759} C_VEL
LIN {X 0,Y 244.892,Z 895.891,A -85,B 0,C 180,E1 -20574.719,E2 -20574.719} C_VEL
LIN {X 0,Y 240.746,Z 906.618,A -85,B 0,C 180,E1 -20576.058,E2 -20576.058} C_VEL
LIN {X 0,Y 236.883,Z 915.763,A -85,B 0,C 180,E1 -20577.467,E2 -20577.467} C_VEL
LIN {X 0,Y 233.741,Z 922.801,A -85,B 0,C 180,E1 -20578.755,E2 -20578.755} C_VEL
LIN {X 0,Y 229.499,Z 931.422,A -85,B 0,C 180,E1 -20580.659,E2 -20580.659} C_VEL
LIN {X 0,Y 225.752,Z 938.836,A -85,B 0,C 180,E1 -20582.662,E2 -20582.662} C_VEL
LIN {X 0,Y 221.932,Z 946.317,A -85,B 0,C 180,E1 -20585.188,E2 -20585.188} C_VEL
LIN {X 0,Y 219.182,Z 951.647,A -85,B 0,C 180,E1 -20587.367,E2 -20587.367} C_VEL
LIN {X 0,Y 216.112,Z 957.778,A -85,B 0,C 180,E1 -20590.576,E2 -20590.576} C_VEL
LIN {X 0,Y 214.146,Z 962.424,A -85,B 0,C 180,E1 -20593.799,E2 -20593.799} C_VEL
LIN {X 0,Y 213.051,Z 965.497,A -85,B 0,C 180,E1 -20596.646,E2 -20596.646} C_VEL
LIN {X 0,Y 212.704,Z 967.118,A -85,B 0,C 180,E1 -20598.563,E2 -20598.563} C_VEL
LIN {X 0,Y 212.835,Z 969.644,A -85,B 0,C 180,E1 -20602.407,E2 -20602.407} C_VEL
LIN {X 0,Y 213.011,Z 971.569,A -85,B 0,C 180,E1 -20604.317,E2 -20604.317} C_VEL
LIN {X 0,Y 213.263,Z 973.005,A -85,B 0,C 180,E1 -20606.218,E2 -20606.218} C_VEL
LIN {X 0,Y 213.506,Z 973.99,A -85,B 0,C 180,E1 -20608.111,E2 -20608.111} C_VEL
LIN {X 0,Y 213.754,Z 974.547,A -85,B 0,C 180,E1 -20609.997,E2 -20609.997} C_VEL
LIN {X 0,Y 213.452,Z 974.596,A -85,B 0,C 180,E1 -20611.884,E2 -20611.884} C_VEL
LIN {X 0,Y 213.195,Z 974.187,A -85,B 0,C 180,E1 -20613.777,E2 -20613.777} C_VEL
LIN {X 0,Y 212.624,Z 972.22,A -85,B 0,C 180,E1 -20617.428,E2 -20617.428} C_VEL
LIN {X 0,Y 212.558,Z 969.44,A -85,B 0,C 180,E1 -20620.475,E2 -20620.475} C_VEL
LIN {X 0,Y 213.019,Z 965.817,A -85,B 0,C 180,E1 -20623.35,E2 -20623.35} C_VEL
LIN {X 0,Y 214.088,Z 961.158,A -85,B 0,C 180,E1 -20626.2,E2 -20626.2} C_VEL
LIN {X 0,Y 215.826,Z 954.888,A -85,B 0,C 180,E1 -20629.207,E2 -20629.207} C_VEL
LIN {X 0,Y 218.036,Z 948.195,A -85,B 0,C 180,E1 -20631.755,E2 -20631.755} C_VEL
LIN {X 0,Y 220.964,Z 939.418,A -85,B 0,C 180,E1 -20634.42,E2 -20634.42} C_VEL
LIN {X 0,Y 223.904,Z 930.49,A -85,B 0,C 180,E1 -20636.566,E2 -20636.566} C_VEL
LIN {X 0,Y 227.258,Z 919.62,A -85,B 0,C 180,E1 -20638.639,E2 -20638.639} C_VEL
LIN {X 0,Y 230.279,Z 908.891,A -85,B 0,C 180,E1 -20640.233,E2 -20640.233} C_VEL
LIN {X 0,Y 233.116,Z 897.005,A -85,B 0,C 180,E1 -20641.586,E2 -20641.586} C_VEL
LIN {X 0,Y 235.369,Z 884.344,A -85,B 0,C 180,E1 -20642.681,E2 -20642.681} C_VEL
LIN {X 0,Y 237.184,Z 870.977,A -85,B 0,C 180,E1 -20643.473,E2 -20643.473} C_VEL
LIN {X 0,Y 238.247,Z 855.614,A -85,B 0,C 180,E1 -20644.032,E2 -20644.032} C_VEL
LIN {X 0,Y 238.912,Z 839.488,A -85,B 0,C 180,E1 -20644.547,E2 -20644.547} C_VEL
LIN {X 0,Y 237.575,Z 815.834,A -85,B 0,C 180,E1 -20645.761,E2 -20645.761} C_VEL
LIN {X 0,Y 235.778,Z 794.179,A -85,B 0,C 180,E1 -20647.033,E2 -20647.033} C_VEL
LIN {X 0,Y 233.537,Z 777.267,A -85,B 0,C 180,E1 -20648.256,E2 -20648.256} C_VEL
LIN {X 0,Y 229.34,Z 767.382,A -85,B 0,C 180,E1 -20649.688,E2 -20649.688} C_VEL
LIN {X 0,Y 226.219,Z 760.904,A -85,B 0,C 180,E1 -20650.778,E2 -20650.778} C_VEL
LIN {X 0,Y 223.932,Z 756.443,A -85,B 0,C 180,E1 -20651.596,E2 -20651.596} C_VEL
LIN {X 0,Y 221.408,Z 751.24,A -85,B 0,C 180,E1 -20652.653,E2 -20652.653} C_VEL
LIN {X 0,Y 219.23,Z 743.084,A -85,B 0,C 180,E1 -20656.43,E2 -20656.43} C_VEL
LIN {X 0,Y 217.36,Z 736.882,A -85,B 0,C 180,E1 -20659.709,E2 -20659.709} C_VEL
LIN {X 0,Y 215.058,Z 729.726,A -85,B 0,C 180,E1 -20663.969,E2 -20663.969} C_VEL
LIN {X 0,Y 213.772,Z 725.893,A -85,B 0,C 180,E1 -20666.728,E2 -20666.728} C_VEL
LIN {X 0,Y 213.771,Z 725.858,A -85,B 0,C 180,E1 -20670.453,E2 -20670.453} C_VEL
LIN {X 0,Y 213.791,Z 725.847,A -85,B 0,C 180,E1 -20674.701,E2 -20674.701} C_VEL
LIN {X 0,Y 213.802,Z 725.843,A -85,B 0,C 180,E1 -20678.803,E2 -20678.803} C_VEL
LIN {X 0,Y 213.933,Z 725.825,A -85,B 0,C 180,E1 -20682.803,E2 -20682.803} C_VEL
LIN {X 0,Y 213.942,Z 725.823,A -85,B 0,C 180,E1 -20686.706,E2 -20686.706} C_VEL
LIN {X 0,Y 214.131,Z 725.798,A -85,B 0,C 180,E1 -20690.555,E2 -20690.555} C_VEL
LIN {X 0,Y 214.197,Z 725.795,A -85,B 0,C 180,E1 -20692.459,E2 -20692.459} C_VEL
LIN {X 0,Y 214.435,Z 725.775,A -85,B 0,C 180,E1 -20698.122,E2 -20698.122} C_VEL
LIN {X 0,Y 214.539,Z 725.747,A -85,B 0,C 180,E1 -20700,E2 -20700} C_VEL
LIN {X 0,Y 214.435,Z 725.77,A -85,B 0,C 180,E1 -20701.878,E2 -20701.878} C_VEL
LIN {X 0,Y 214.217,Z 725.795,A -85,B 0,C 180,E1 -20707.541,E2 -20707.541} C_VEL
LIN {X 0,Y 214.013,Z 725.822,A -85,B 0,C 180,E1 -20711.364,E2 -20711.364} C_VEL
LIN {X 0,Y 213.923,Z 725.831,A -85,B 0,C 180,E1 -20715.238,E2 -20715.238} C_VEL
LIN {X 0,Y 213.825,Z 725.842,A -85,B 0,C 180,E1 -20719.189,E2 -20719.189} C_VEL
LIN {X 0,Y 213.872,Z 726.102,A -85,B 0,C 180,E1 -20720.561,E2 -20720.561} C_VEL
LIN {X 0,Y 214.183,Z 727.381,A -85,B 0,C 180,E1 -20721.033,E2 -20721.033} C_VEL
LIN {X 0,Y 215.801,Z 729.987,A -85,B 0,C 180,E1 -20721.744,E2 -20721.744} C_VEL
LIN {X 0,Y 217.396,Z 731.455,A -85,B 0,C 180,E1 -20722.337,E2 -20722.337} C_VEL
LIN {X 0,Y 219.469,Z 734.724,A -85,B 0,C 180,E1 -20723.159,E2 -20723.159} C_VEL
LIN {X 0,Y 221.031,Z 736.64,A -85,B 0,C 180,E1 -20723.73,E2 -20723.73} C_VEL
LIN {X 0,Y 226.973,Z 745.273,A -85,B 0,C 180,E1 -20725.816,E2 -20725.816} C_VEL
LIN {X 0,Y 233.514,Z 755.853,A -85,B 0,C 180,E1 -20727.93,E2 -20727.93} C_VEL
LIN {X 0,Y 239.522,Z 766.802,A -85,B 0,C 180,E1 -20729.746,E2 -20729.746} C_VEL
LIN {X 0,Y 242.116,Z 772.092,A -85,B 0,C 180,E1 -20730.501,E2 -20730.501} C_VEL
LIN {X 0,Y 240.837,Z 806.45,A -85,B 0,C 180,E1 -20731.641,E2 -20731.641} C_VEL
LIN {X 0,Y 240.326,Z 819.714,A -85,B 0,C 180,E1 -20732.26,E2 -20732.26} C_VEL
LIN {X 0,Y 239.289,Z 832.307,A -85,B 0,C 180,E1 -20733.176,E2 -20733.176} C_VEL
LIN {X 0,Y 237.574,Z 844.96,A -85,B 0,C 180,E1 -20734.426,E2 -20734.426} C_VEL
LIN {X 0,Y 235.429,Z 856.439,A -85,B 0,C 180,E1 -20735.935,E2 -20735.935} C_VEL
LIN {X 0,Y 232.864,Z 867.398,A -85,B 0,C 180,E1 -20737.776,E2 -20737.776} C_VEL
LIN {X 0,Y 230.104,Z 877.34,A -85,B 0,C 180,E1 -20739.897,E2 -20739.897} C_VEL
LIN {X 0,Y 227.43,Z 885.657,A -85,B 0,C 180,E1 -20742.133,E2 -20742.133} C_VEL
LIN {X 0,Y 224.705,Z 893.15,A -85,B 0,C 180,E1 -20744.644,E2 -20744.644} C_VEL
LIN {X 0,Y 222.29,Z 899.436,A -85,B 0,C 180,E1 -20747.336,E2 -20747.336} C_VEL
LIN {X 0,Y 219.964,Z 904.754,A -85,B 0,C 180,E1 -20750.286,E2 -20750.286} C_VEL
LIN {X 0,Y 217.747,Z 909.258,A -85,B 0,C 180,E1 -20753.795,E2 -20753.795} C_VEL
LIN {X 0,Y 216.068,Z 912.358,A -85,B 0,C 180,E1 -20757.748,E2 -20757.748} C_VEL
LIN {X 0,Y 215.233,Z 913.465,A -85,B 0,C 180,E1 -20760.676,E2 -20760.676} C_VEL
LIN {X 0,Y 214.859,Z 913.665,A -85,B 0,C 180,E1 -20762.749,E2 -20762.749} C_VEL
LIN {X 0,Y 214.663,Z 913.412,A -85,B 0,C 180,E1 -20764.814,E2 -20764.814} C_VEL
LIN {X 0,Y 214.636,Z 912.651,A -85,B 0,C 180,E1 -20766.867,E2 -20766.867} C_VEL
LIN {X 0,Y 214.784,Z 911.459,A -85,B 0,C 180,E1 -20768.907,E2 -20768.907} C_VEL
LIN {X 0,Y 215.174,Z 909.423,A -85,B 0,C 180,E1 -20771.299,E2 -20771.299} C_VEL
LIN {X 0,Y 216.31,Z 904.976,A -85,B 0,C 180,E1 -20774.938,E2 -20774.938} C_VEL
LIN {X 0,Y 217.535,Z 899.984,A -85,B 0,C 180,E1 -20777.881,E2 -20777.881} C_VEL
LIN {X 0,Y 219.17,Z 893.625,A -85,B 0,C 180,E1 -20780.777,E2 -20780.777} C_VEL
LIN {X 0,Y 221.123,Z 885.729,A -85,B 0,C 180,E1 -20783.616,E2 -20783.616} C_VEL
LIN {X 0,Y 222.972,Z 877.674,A -85,B 0,C 180,E1 -20785.936,E2 -20785.936} C_VEL
LIN {X 0,Y 225.048,Z 867.802,A -85,B 0,C 180,E1 -20788.213,E2 -20788.213} C_VEL
LIN {X 0,Y 227.06,Z 856.873,A -85,B 0,C 180,E1 -20790.224,E2 -20790.224} C_VEL
LIN {X 0,Y 228.693,Z 846.342,A -85,B 0,C 180,E1 -20791.764,E2 -20791.764} C_VEL
LIN {X 0,Y 230.108,Z 834.903,A -85,B 0,C 180,E1 -20793.066,E2 -20793.066} C_VEL
LIN {X 0,Y 231.186,Z 821.618,A -85,B 0,C 180,E1 -20794.197,E2 -20794.197} C_VEL
LIN {X 0,Y 231.801,Z 808.518,A -85,B 0,C 180,E1 -20794.949,E2 -20794.949} C_VEL
LIN {X 0,Y 232.681,Z 772.49,A -85,B 0,C 180,E1 -20796.166,E2 -20796.166} C_VEL
LIN {X 0,Y 232.977,Z 764.13,A -85,B 0,C 180,E1 -20796.429,E2 -20796.429} C_VEL
LIN {X 0,Y 227.734,Z 752.678,A -85,B 0,C 180,E1 -20797.563,E2 -20797.563} C_VEL
LIN {X 0,Y 218.801,Z 735.114,A -85,B 0,C 180,E1 -20799.57,E2 -20799.57} C_VEL
LIN {X 0,Y 215.201,Z 728.836,A -85,B 0,C 180,E1 -20800.399,E2 -20800.399} C_VEL
LIN {X 0,Y 214.136,Z 726.405,A -85,B 0,C 180,E1 -20800.802,E2 -20800.802} C_VEL
LIN {X 0,Y 213.995,Z 725.84,A -85,B 0,C 180,E1 -20801.367,E2 -20801.367} C_VEL
LIN {X 0,Y 213.888,Z 725.826,A -85,B 0,C 180,E1 -20805.243,E2 -20805.243} C_VEL
LIN {X 0,Y 213.798,Z 725.834,A -85,B 0,C 180,E1 -20809.194,E2 -20809.194} C_VEL
LIN {X 0,Y 213.79,Z 725.856,A -85,B 0,C 180,E1 -20813.236,E2 -20813.236} C_VEL
LIN {X 0,Y 213.773,Z 725.828,A -85,B 0,C 180,E1 -20817.419,E2 -20817.419} C_VEL
LIN {X 0,Y 213.765,Z 725.851,A -85,B 0,C 180,E1 -20821.741,E2 -20821.741} C_VEL
LIN {X 0,Y 213.747,Z 725.824,A -85,B 0,C 180,E1 -20826.291,E2 -20826.291} C_VEL
LIN {X 0,Y 213.705,Z 725.866,A -85,B 0,C 180,E1 -20831.13,E2 -20831.13} C_VEL
LIN {X 0,Y 213.709,Z 725.866,A -85,B 0,C 180,E1 -20833.681,E2 -20833.681} C_VEL
LIN {X 0,Y 213.743,Z 725.962,A -85,B 0,C 180,E1 -20837.982,E2 -20837.982} C_VEL
LIN {X 0,Y 213.927,Z 726.826,A -85,B 0,C 180,E1 -20838.324,E2 -20838.324} C_VEL
LIN {X 0,Y 223.788,Z 755.37,A -85,B 0,C 180,E1 -20840.483,E2 -20840.483} C_VEL
LIN {X 0,Y 221.908,Z 806.398,A -85,B 0,C 180,E1 -20842.881,E2 -20842.881} C_VEL
LIN {X 0,Y 221.502,Z 817.271,A -85,B 0,C 180,E1 -20843.634,E2 -20843.634} C_VEL
LIN {X 0,Y 220.735,Z 828.108,A -85,B 0,C 180,E1 -20844.614,E2 -20844.614} C_VEL
LIN {X 0,Y 219.945,Z 837.991,A -85,B 0,C 180,E1 -20845.736,E2 -20845.736} C_VEL
LIN {X 0,Y 219.147,Z 846.95,A -85,B 0,C 180,E1 -20846.962,E2 -20846.962} C_VEL
LIN {X 0,Y 218.108,Z 857.376,A -85,B 0,C 180,E1 -20848.695,E2 -20848.695} C_VEL
LIN {X 0,Y 217.19,Z 866.102,A -85,B 0,C 180,E1 -20850.431,E2 -20850.431} C_VEL
LIN {X 0,Y 216.476,Z 872.62,A -85,B 0,C 180,E1 -20851.916,E2 -20851.916} C_VEL
LIN {X 0,Y 215.453,Z 881.679,A -85,B 0,C 180,E1 -20854.392,E2 -20854.392} C_VEL
LIN {X 0,Y 214.964,Z 887.561,A -85,B 0,C 180,E1 -20856.272,E2 -20856.272} C_VEL
LIN {X 0,Y 214.383,Z 894.336,A -85,B 0,C 180,E1 -20858.862,E2 -20858.862} C_VEL
LIN {X 0,Y 214.143,Z 898.761,A -85,B 0,C 180,E1 -20860.84,E2 -20860.84} C_VEL
LIN {X 0,Y 213.994,Z 904.047,A -85,B 0,C 180,E1 -20863.79,E2 -20863.79} C_VEL
LIN {X 0,Y 214.247,Z 908.118,A -85,B 0,C 180,E1 -20866.725,E2 -20866.725} C_VEL
LIN {X 0,Y 214.713,Z 910.695,A -85,B 0,C 180,E1 -20869.114,E2 -20869.114} C_VEL
